LIN {X 0,Y 467.565,Z 337.401,A -85,B 0,C 180,E1 -7610.122,E2 -7610.122} C_VEL
LIN {X 0,Y 469.367,Z 346.484,A -85,B 0,C 180,E1 -7612.893,E2 -7612.893} C_VEL
LIN {X 0,Y 469.775,Z 350.018,A -85,B 0,C 180,E1 -7613.888,E2 -7613.888} C_VEL
LIN {X 0,Y 468.945,Z 363.418,A -85,B 0,C 180,E1 -7617.35,E2 -7617.35} C_VEL
LIN {X 0,Y 468.563,Z 374.519,A -85,B 0,C 180,E1 -7620.086,E2 -7620.086} C_VEL
LIN {X 0,Y 468.19,Z 387.799,A -85,B 0,C 180,E1 -7623.236,E2 -7623.236} C_VEL
LIN {X 0,Y 467.873,Z 401.533,A -85,B 0,C 180,E1 -7626.39,E2 -7626.39} C_VEL
LIN {X 0,Y 467.562,Z 416.649,A -85,B 0,C 180,E1 -7629.775,E2 -7629.775} C_VEL
LIN {X 0,Y 467.339,Z 431.071,A -85,B 0,C 180,E1 -7632.948,E2 -7632.948} C_VEL
LIN {X 0,Y 467.254,Z 438.483,A -85,B 0,C 180,E1 -7634.516,E2 -7634.516} C_VEL
LIN {X 0,Y 467.458,Z 441.247,A -85,B 0,C 180,E1 -7634.62,E2 -7634.62} C_VEL
LIN {X 0,Y 468.524,Z 455.112,A -85,B 0,C 180,E1 -7635.032,E2 -7635.032} C_VEL
LIN {X 0,Y 469.497,Z 465.721,A -85,B 0,C 180,E1 -7635.479,E2 -7635.479} C_VEL
LIN {X 0,Y 469.015,Z 478.326,A -85,B 0,C 180,E1 -7636.128,E2 -7636.128} C_VEL
LIN {X 0,Y 468.559,Z 489.635,A -85,B 0,C 180,E1 -7636.888,E2 -7636.888} C_VEL
LIN {X 0,Y 468.224,Z 499.908,A -85,B 0,C 180,E1 -7637.742,E2 -7637.742} C_VEL
LIN {X 0,Y 467.755,Z 509.75,A -85,B 0,C 180,E1 -7638.737,E2 -7638.737} C_VEL
LIN {X 0,Y 467.388,Z 518.626,A -85,B 0,C 180,E1 -7639.824,E2 -7639.824} C_VEL
LIN {X 0,Y 467.148,Z 527.303,A -85,B 0,C 180,E1 -7641.129,E2 -7641.129} C_VEL
LIN {X 0,Y 467.045,Z 534.318,A -85,B 0,C 180,E1 -7642.434,E2 -7642.434} C_VEL
LIN {X 0,Y 467.012,Z 540.786,A -85,B 0,C 180,E1 -7643.953,E2 -7643.953} C_VEL
LIN {X 0,Y 466.979,Z 544.992,A -85,B 0,C 180,E1 -7645.252,E2 -7645.252} C_VEL
LIN {X 0,Y 466.988,Z 548.116,A -85,B 0,C 180,E1 -7646.549,E2 -7646.549} C_VEL
LIN {X 0,Y 466.982,Z 549.617,A -85,B 0,C 180,E1 -7647.412,E2 -7647.412} C_VEL
LIN {X 0,Y 467.076,Z 551.385,A -85,B 0,C 180,E1 -7649.138,E2 -7649.138} C_VEL
LIN {X 0,Y 467.064,Z 551.647,A -85,B 0,C 180,E1 -7650,E2 -7650} C_VEL
LIN {X 0,Y 467.075,Z 551.459,A -85,B 0,C 180,E1 -7650.862,E2 -7650.862} C_VEL
LIN {X 0,Y 466.955,Z 549.855,A -85,B 0,C 180,E1 -7652.588,E2 -7652.588} C_VEL
LIN {X 0,Y 466.966,Z 548.427,A -85,B 0,C 180,E1 -7653.451,E2 -7653.451} C_VEL
LIN {X 0,Y 466.951,Z 545.43,A -85,B 0,C 180,E1 -7654.748,E2 -7654.748} C_VEL
LIN {X 0,Y 466.971,Z 540.24,A -85,B 0,C 180,E1 -7656.343,E2 -7656.343} C_VEL
LIN {X 0,Y 467.03,Z 534.045,A -85,B 0,C 180,E1 -7657.784,E2 -7657.784} C_VEL
LIN {X 0,Y 467.175,Z 526.937,A -85,B 0,C 180,E1 -7659.088,E2 -7659.088} C_VEL
LIN {X 0,Y 467.453,Z 518.079,A -85,B 0,C 180,E1 -7660.394,E2 -7660.394} C_VEL
LIN {X 0,Y 467.832,Z 509.046,A -85,B 0,C 180,E1 -7661.481,E2 -7661.481} C_VEL
LIN {X 0,Y 468.296,Z 499.714,A -85,B 0,C 180,E1 -7662.406,E2 -7662.406} C_VEL
LIN {X 0,Y 468.724,Z 488.228,A -85,B 0,C 180,E1 -7663.328,E2 -7663.328} C_VEL
LIN {X 0,Y 469.261,Z 476.177,A -85,B 0,C 180,E1 -7664.085,E2 -7664.085} C_VEL
LIN {X 0,Y 469.619,Z 464.972,A -85,B 0,C 180,E1 -7664.627,E2 -7664.627} C_VEL
LIN {X 0,Y 468.446,Z 452.922,A -85,B 0,C 180,E1 -7665.096,E2 -7665.096} C_VEL
LIN {X 0,Y 467.289,Z 441.274,A -85,B 0,C 180,E1 -7665.427,E2 -7665.427} C_VEL
LIN {X 0,Y 467.275,Z 440.651,A -85,B 0,C 180,E1 -7665.483,E2 -7665.483} C_VEL
LIN {X 0,Y 467.587,Z 425.096,A -85,B 0,C 180,E1 -7668.974,E2 -7668.974} C_VEL
LIN {X 0,Y 468,Z 409.645,A -85,B 0,C 180,E1 -7672.515,E2 -7672.515} C_VEL
LIN {X 0,Y 468.463,Z 395.511,A -85,B 0,C 180,E1 -7675.824,E2 -7675.824} C_VEL
LIN {X 0,Y 468.898,Z 382.637,A -85,B 0,C 180,E1 -7678.905,E2 -7678.905} C_VEL
LIN {X 0,Y 469.437,Z 370.623,A -85,B 0,C 180,E1 -7681.851,E2 -7681.851} C_VEL
LIN {X 0,Y 470.388,Z 355.622,A -85,B 0,C 180,E1 -7685.639,E2 -7685.639} C_VEL
LIN {X 0,Y 470.406,Z 351.582,A -85,B 0,C 180,E1 -7686.698,E2 -7686.698} C_VEL
LIN {X 0,Y 468.436,Z 341.626,A -85,B 0,C 180,E1 -7689.523,E2 -7689.523} C_VEL
LIN {X 0,Y 467.561,Z 337.324,A -85,B 0,C 180,E1 -7690.832,E2 -7690.832} C_VEL
LIN {X 0,Y 467.539,Z 337.249,A -85,B 0,C 180,E1 -7693.819,E2 -7693.819} C_VEL
LIN {X 0,Y 467.54,Z 337.245,A -85,B 0,C 180,E1 -7696.254,E2 -7696.254} C_VEL
LIN {X 0,Y 467.551,Z 337.244,A -85,B 0,C 180,E1 -7699.732,E2 -7699.732} C_VEL
LIN {X 0,Y 467.54,Z 337.244,A -85,B 0,C 180,E1 -7702.813,E2 -7702.813} C_VEL
LIN {X 0,Y 467.569,Z 337.24,A -85,B 0,C 180,E1 -7705.759,E2 -7705.759} C_VEL
LIN {X 0,Y 467.559,Z 337.243,A -85,B 0,C 180,E1 -7708.955,E2 -7708.955} C_VEL
LIN {X 0,Y 467.625,Z 337.232,A -85,B 0,C 180,E1 -7712.461,E2 -7712.461} C_VEL
LIN {X 0,Y 467.576,Z 337.245,A -85,B 0,C 180,E1 -7715.111,E2 -7715.111} C_VEL
LIN {X 0,Y 467.524,Z 337.244,A -85,B 0,C 180,E1 -7717.926,E2 -7717.926} C_VEL
LIN {X 0,Y 467.612,Z 337.236,A -85,B 0,C 180,E1 -7720.692,E2 -7720.692} C_VEL
LIN {X 0,Y 467.628,Z 337.231,A -85,B 0,C 180,E1 -7724.305,E2 -7724.305} C_VEL
LIN {X 0,Y 467.645,Z 337.228,A -85,B 0,C 180,E1 -7727.854,E2 -7727.854} C_VEL
LIN {X 0,Y 467.659,Z 337.229,A -85,B 0,C 180,E1 -7731.357,E2 -7731.357} C_VEL
LIN {X 0,Y 467.722,Z 337.219,A -85,B 0,C 180,E1 -7733.962,E2 -7733.962} C_VEL
LIN {X 0,Y 467.846,Z 337.205,A -85,B 0,C 180,E1 -7737.417,E2 -7737.417} C_VEL
LIN {X 0,Y 467.869,Z 337.201,A -85,B 0,C 180,E1 -7740,E2 -7740} C_VEL
LIN {X 0,Y 467.847,Z 337.209,A -85,B 0,C 180,E1 -7742.583,E2 -7742.583} C_VEL
LIN {X 0,Y 467.723,Z 337.22,A -85,B 0,C 180,E1 -7746.038,E2 -7746.038} C_VEL
LIN {X 0,Y 467.671,Z 337.233,A -85,B 0,C 180,E1 -7748.643,E2 -7748.643} C_VEL
LIN {X 0,Y 467.646,Z 337.231,A -85,B 0,C 180,E1 -7752.146,E2 -7752.146} C_VEL
LIN {X 0,Y 467.629,Z 337.23,A -85,B 0,C 180,E1 -7755.695,E2 -7755.695} C_VEL
LIN {X 0,Y 467.608,Z 337.238,A -85,B 0,C 180,E1 -7758.765,E2 -7758.765} C_VEL
LIN {X 0,Y 467.575,Z 337.238,A -85,B 0,C 180,E1 -7761.27,E2 -7761.27} C_VEL
LIN {X 0,Y 467.567,Z 337.24,A -85,B 0,C 180,E1 -7763.944,E2 -7763.944} C_VEL
LIN {X 0,Y 467.608,Z 337.236,A -85,B 0,C 180,E1 -7766.801,E2 -7766.801} C_VEL
LIN {X 0,Y 467.579,Z 337.238,A -85,B 0,C 180,E1 -7769.736,E2 -7769.736} C_VEL
LIN {X 0,Y 467.576,Z 337.24,A -85,B 0,C 180,E1 -7772.759,E2 -7772.759} C_VEL
LIN {X 0,Y 467.549,Z 337.243,A -85,B 0,C 180,E1 -7775.89,E2 -7775.89} C_VEL
LIN {X 0,Y 467.591,Z 337.235,A -85,B 0,C 180,E1 -7779.144,E2 -7779.144} C_VEL
LIN {X 0,Y 467.581,Z 337.24,A -85,B 0,C 180,E1 -7782.568,E2 -7782.568} C_VEL
LIN {X 0,Y 467.566,Z 337.238,A -85,B 0,C 180,E1 -7785.054,E2 -7785.054} C_VEL
LIN {X 0,Y 467.585,Z 337.237,A -85,B 0,C 180,E1 -7787.441,E2 -7787.441} C_VEL
LIN {X 0,Y 467.578,Z 337.237,A -85,B 0,C 180,E1 -7790.856,E2 -7790.856} C_VEL
LIN {X 0,Y 467.56,Z 337.244,A -85,B 0,C 180,E1 -7794.261,E2 -7794.261} C_VEL
LIN {X 0,Y 467.58,Z 337.237,A -85,B 0,C 180,E1 -7797.322,E2 -7797.322} C_VEL
LIN {X 0,Y 467.578,Z 337.237,A -85,B 0,C 180,E1 -7800.666,E2 -7800.666} C_VEL
LIN {X 0,Y 467.628,Z 337.231,A -85,B 0,C 180,E1 -7803.201,E2 -7803.201} C_VEL
LIN {X 0,Y 467.594,Z 337.236,A -85,B 0,C 180,E1 -7806.469,E2 -7806.469} C_VEL
LIN {X 0,Y 467.625,Z 337.239,A -85,B 0,C 180,E1 -7809.778,E2 -7809.778} C_VEL
LIN {X 0,Y 467.61,Z 337.233,A -85,B 0,C 180,E1 -7812.507,E2 -7812.507} C_VEL
LIN {X 0,Y 467.608,Z 337.235,A -85,B 0,C 180,E1 -7815.197,E2 -7815.197} C_VEL
LIN {X 0,Y 467.599,Z 337.235,A -85,B 0,C 180,E1 -7815.441,E2 -7815.441} C_VEL
LIN {X 0,Y 466.929,Z 337.321,A -85,B 0,C 180,E1 -7816.16,E2 -7816.16} C_VEL
LIN {X 0,Y 464.085,Z 337.675,A -85,B 0,C 180,E1 -7817.329,E2 -7817.329} C_VEL
LIN {X 0,Y 461.686,Z 337.972,A -85,B 0,C 180,E1 -7818.271,E2 -7818.271} C_VEL
LIN {X 0,Y 460.661,Z 338.099,A -85,B 0,C 180,E1 -7818.998,E2 -7818.998} C_VEL
LIN {X 0,Y 460.58,Z 338.111,A -85,B 0,C 180,E1 -7819.245,E2 -7819.245} C_VEL
LIN {X 0,Y 460.723,Z 338.091,A -85,B 0,C 180,E1 -7822.538,E2 -7822.538} C_VEL
LIN {X 0,Y 460.702,Z 338.093,A -85,B 0,C 180,E1 -7824.749,E2 -7824.749} C_VEL
LIN {X 0,Y 460.828,Z 338.083,A -85,B 0,C 180,E1 -7827.378,E2 -7827.378} C_VEL
LIN {X 0,Y 460.857,Z 338.077,A -85,B 0,C 180,E1 -7830,E2 -7830} C_VEL
LIN {X 0,Y 460.828,Z 338.078,A -85,B 0,C 180,E1 -7832.622,E2 -7832.622} C_VEL
LIN {X 0,Y 460.704,Z 338.094,A -85,B 0,C 180,E1 -7836.13,E2 -7836.13} C_VEL
LIN {X 0,Y 460.631,Z 338.103,A -85,B 0,C 180,E1 -7838.776,E2 -7838.776} C_VEL
LIN {X 0,Y 460.615,Z 338.104,A -85,B 0,C 180,E1 -7842.445,E2 -7842.445} C_VEL
LIN {X 0,Y 460.602,Z 338.107,A -85,B 0,C 180,E1 -7845.997,E2 -7845.997} C_VEL
LIN {X 0,Y 460.573,Z 338.113,A -85,B 0,C 180,E1 -7848.902,E2 -7848.902} C_VEL
LIN {X 0,Y 460.517,Z 338.121,A -85,B 0,C 180,E1 -7851.485,E2 -7851.485} C_VEL
LIN {X 0,Y 460.543,Z 338.113,A -85,B 0,C 180,E1 -7854.332,E2 -7854.332} C_VEL
LIN {X 0,Y 460.584,Z 338.115,A -85,B 0,C 180,E1 -7857.242,E2 -7857.242} C_VEL
LIN {X 0,Y 460.51,Z 338.117,A -85,B 0,C 180,E1 -7860.239,E2 -7860.239} C_VEL
LIN {X 0,Y 460.528,Z 338.12,A -85,B 0,C 180,E1 -7863.324,E2 -7863.324} C_VEL
LIN {X 0,Y 460.479,Z 338.123,A -85,B 0,C 180,E1 -7866.528,E2 -7866.528} C_VEL
LIN {X 0,Y 460.576,Z 338.111,A -85,B 0,C 180,E1 -7869.857,E2 -7869.857} C_VEL
LIN {X 0,Y 460.539,Z 338.121,A -85,B 0,C 180,E1 -7872.904,E2 -7872.904} C_VEL
LIN {X 0,Y 460.519,Z 338.121,A -85,B 0,C 180,E1 -7875.828,E2 -7875.828} C_VEL
LIN {X 0,Y 460.635,Z 338.281,A -85,B 0,C 180,E1 -7877.236,E2 -7877.236} C_VEL
LIN {X 0,Y 460.785,Z 339.139,A -85,B 0,C 180,E1 -7877.371,E2 -7877.371} C_VEL
LIN {X 0,Y 463.382,Z 348.732,A -85,B 0,C 180,E1 -7878.001,E2 -7878.001} C_VEL
LIN {X 0,Y 462.957,Z 360.559,A -85,B 0,C 180,E1 -7878.817,E2 -7878.817} C_VEL
LIN {X 0,Y 462.47,Z 371.478,A -85,B 0,C 180,E1 -7879.77,E2 -7879.77} C_VEL
LIN {X 0,Y 462.064,Z 381.585,A -85,B 0,C 180,E1 -7880.868,E2 -7880.868} C_VEL
LIN {X 0,Y 461.625,Z 389.546,A -85,B 0,C 180,E1 -7881.923,E2 -7881.923} C_VEL
LIN {X 0,Y 461.224,Z 397.793,A -85,B 0,C 180,E1 -7883.267,E2 -7883.267} C_VEL
LIN {X 0,Y 460.926,Z 404.327,A -85,B 0,C 180,E1 -7884.591,E2 -7884.591} C_VEL
LIN {X 0,Y 460.623,Z 410.341,A -85,B 0,C 180,E1 -7886.158,E2 -7886.158} C_VEL
LIN {X 0,Y 460.442,Z 414.737,A -85,B 0,C 180,E1 -7887.709,E2 -7887.709} C_VEL
LIN {X 0,Y 460.369,Z 416.902,A -85,B 0,C 180,E1 -7888.746,E2 -7888.746} C_VEL
LIN {X 0,Y 460.222,Z 419.248,A -85,B 0,C 180,E1 -7890.507,E2 -7890.507} C_VEL
LIN {X 0,Y 460.209,Z 419.967,A -85,B 0,C 180,E1 -7892.34,E2 -7892.34} C_VEL
LIN {X 0,Y 460.319,Z 418.895,A -85,B 0,C 180,E1 -7894.26,E2 -7894.26} C_VEL
LIN {X 0,Y 460.457,Z 416.885,A -85,B 0,C 180,E1 -7895.663,E2 -7895.663} C_VEL
LIN {X 0,Y 460.657,Z 413.689,A -85,B 0,C 180,E1 -7897.105,E2 -7897.105} C_VEL
LIN {X 0,Y 460.883,Z 409.313,A -85,B 0,C 180,E1 -7898.532,E2 -7898.532} C_VEL
LIN {X 0,Y 461.218,Z 403.626,A -85,B 0,C 180,E1 -7899.949,E2 -7899.949} C_VEL
LIN {X 0,Y 461.631,Z 396.366,A -85,B 0,C 180,E1 -7901.355,E2 -7901.355} C_VEL
LIN {X 0,Y 462.119,Z 387.293,A -85,B 0,C 180,E1 -7902.749,E2 -7902.749} C_VEL
LIN {X 0,Y 462.661,Z 377.58,A -85,B 0,C 180,E1 -7903.926,E2 -7903.926} C_VEL
LIN {X 0,Y 463.097,Z 367.275,A -85,B 0,C 180,E1 -7904.936,E2 -7904.936} C_VEL
LIN {X 0,Y 463.511,Z 356.547,A -85,B 0,C 180,E1 -7905.779,E2 -7905.779} C_VEL
LIN {X 0,Y 463.584,Z 348.504,A -85,B 0,C 180,E1 -7906.298,E2 -7906.298} C_VEL
LIN {X 0,Y 460.717,Z 338.858,A -85,B 0,C 180,E1 -7906.958,E2 -7906.958} C_VEL
LIN {X 0,Y 460.583,Z 338.152,A -85,B 0,C 180,E1 -7907.139,E2 -7907.139} C_VEL
LIN {X 0,Y 460.577,Z 338.116,A -85,B 0,C 180,E1 -7909.449,E2 -7909.449} C_VEL
LIN {X 0,Y 460.704,Z 338.097,A -85,B 0,C 180,E1 -7912.543,E2 -7912.543} C_VEL
LIN {X 0,Y 460.682,Z 338.101,A -85,B 0,C 180,E1 -7914.748,E2 -7914.748} C_VEL
LIN {X 0,Y 460.788,Z 338.089,A -85,B 0,C 180,E1 -7917.377,E2 -7917.377} C_VEL
LIN {X 0,Y 460.84,Z 338.079,A -85,B 0,C 180,E1 -7920,E2 -7920} C_VEL
LIN {X 0,Y 460.788,Z 338.086,A -85,B 0,C 180,E1 -7922.623,E2 -7922.623} C_VEL
LIN {X 0,Y 460.687,Z 338.097,A -85,B 0,C 180,E1 -7926.13,E2 -7926.13} C_VEL
LIN {X 0,Y 460.609,Z 338.109,A -85,B 0,C 180,E1 -7928.777,E2 -7928.777} C_VEL
LIN {X 0,Y 460.598,Z 338.107,A -85,B 0,C 180,E1 -7932.335,E2 -7932.335} C_VEL
LIN {X 0,Y 460.591,Z 338.109,A -85,B 0,C 180,E1 -7935.998,E2 -7935.998} C_VEL
LIN {X 0,Y 460.558,Z 338.113,A -85,B 0,C 180,E1 -7939.616,E2 -7939.616} C_VEL
LIN {X 0,Y 460.501,Z 338.122,A -85,B 0,C 180,E1 -7942.429,E2 -7942.429} C_VEL
LIN {X 0,Y 460.545,Z 338.113,A -85,B 0,C 180,E1 -7945.799,E2 -7945.799} C_VEL
LIN {X 0,Y 460.543,Z 338.116,A -85,B 0,C 180,E1 -7948.234,E2 -7948.234} C_VEL
LIN {X 0,Y 460.512,Z 338.122,A -85,B 0,C 180,E1 -7951.283,E2 -7951.283} C_VEL
LIN {X 0,Y 460.515,Z 338.122,A -85,B 0,C 180,E1 -7954.504,E2 -7954.504} C_VEL
LIN {X 0,Y 460.493,Z 338.123,A -85,B 0,C 180,E1 -7957.624,E2 -7957.624} C_VEL
LIN {X 0,Y 460.509,Z 338.124,A -85,B 0,C 180,E1 -7961.014,E2 -7961.014} C_VEL
LIN {X 0,Y 460.506,Z 338.121,A -85,B 0,C 180,E1 -7964.59,E2 -7964.59} C_VEL
LIN {X 0,Y 460.486,Z 338.124,A -85,B 0,C 180,E1 -7967.816,E2 -7967.816} C_VEL
LIN {X 0,Y 460.534,Z 338.278,A -85,B 0,C 180,E1 -7969.808,E2 -7969.808} C_VEL
LIN {X 0,Y 462.265,Z 347.022,A -85,B 0,C 180,E1 -7972.546,E2 -7972.546} C_VEL
LIN {X 0,Y 462.809,Z 350.922,A -85,B 0,C 180,E1 -7973.685,E2 -7973.685} C_VEL
LIN {X 0,Y 462.069,Z 362.679,A -85,B 0,C 180,E1 -7976.802,E2 -7976.802} C_VEL
LIN {X 0,Y 461.581,Z 374.697,A -85,B 0,C 180,E1 -7979.838,E2 -7979.838} C_VEL
LIN {X 0,Y 461.162,Z 387.905,A -85,B 0,C 180,E1 -7983.04,E2 -7983.04} C_VEL
LIN {X 0,Y 460.8,Z 401.493,A -85,B 0,C 180,E1 -7986.221,E2 -7986.221} C_VEL
LIN {X 0,Y 460.528,Z 415.613,A -85,B 0,C 180,E1 -7989.452,E2 -7989.452} C_VEL
LIN {X 0,Y 460.278,Z 429.983,A -85,B 0,C 180,E1 -7992.678,E2 -7992.678} C_VEL
LIN {X 0,Y 460.201,Z 437.169,A -85,B 0,C 180,E1 -7994.239,E2 -7994.239} C_VEL
LIN {X 0,Y 460.353,Z 439.549,A -85,B 0,C 180,E1 -7994.356,E2 -7994.356} C_VEL
LIN {X 0,Y 461.551,Z 454.098,A -85,B 0,C 180,E1 -7994.798,E2 -7994.798} C_VEL
LIN {X 0,Y 462.484,Z 467.088,A -85,B 0,C 180,E1 -7995.367,E2 -7995.367} C_VEL
LIN {X 0,Y 461.995,Z 478.993,A -85,B 0,C 180,E1 -7996.026,E2 -7996.026} C_VEL
LIN {X 0,Y 461.521,Z 489.961,A -85,B 0,C 180,E1 -7996.796,E2 -7996.796} C_VEL
LIN {X 0,Y 461.166,Z 500.175,A -85,B 0,C 180,E1 -7997.681,E2 -7997.681} C_VEL
LIN {X 0,Y 460.677,Z 508.638,A -85,B 0,C 180,E1 -7998.561,E2 -7998.561} C_VEL
LIN {X 0,Y 460.329,Z 517.532,A -85,B 0,C 180,E1 -7999.666,E2 -7999.666} C_VEL
LIN {X 0,Y 460.093,Z 526.222,A -85,B 0,C 180,E1 -8000.992,E2 -8000.992} C_VEL
LIN {X 0,Y 459.988,Z 533.25,A -85,B 0,C 180,E1 -8002.317,E2 -8002.317} C_VEL
LIN {X 0,Y 459.957,Z 539.734,A -85,B 0,C 180,E1 -8003.86,E2 -8003.86} C_VEL
LIN {X 0,Y 459.935,Z 543.956,A -85,B 0,C 180,E1 -8005.179,E2 -8005.179} C_VEL
LIN {X 0,Y 459.943,Z 547.093,A -85,B 0,C 180,E1 -8006.496,E2 -8006.496} C_VEL
LIN {X 0,Y 459.941,Z 548.602,A -85,B 0,C 180,E1 -8007.373,E2 -8007.373} C_VEL
LIN {X 0,Y 460.058,Z 550.388,A -85,B 0,C 180,E1 -8009.125,E2 -8009.125} C_VEL
LIN {X 0,Y 460.047,Z 550.654,A -85,B 0,C 180,E1 -8010,E2 -8010} C_VEL
LIN {X 0,Y 460.055,Z 550.469,A -85,B 0,C 180,E1 -8010.875,E2 -8010.875} C_VEL
LIN {X 0,Y 459.911,Z 548.868,A -85,B 0,C 180,E1 -8012.628,E2 -8012.628} C_VEL
LIN {X 0,Y 459.922,Z 547.439,A -85,B 0,C 180,E1 -8013.504,E2 -8013.504} C_VEL
LIN {X 0,Y 459.901,Z 544.441,A -85,B 0,C 180,E1 -8014.821,E2 -8014.821} C_VEL
LIN {X 0,Y 459.916,Z 540.361,A -85,B 0,C 180,E1 -8016.14,E2 -8016.14} C_VEL
LIN {X 0,Y 459.944,Z 534.065,A -85,B 0,C 180,E1 -8017.683,E2 -8017.683} C_VEL
LIN {X 0,Y 460.062,Z 527.212,A -85,B 0,C 180,E1 -8019.008,E2 -8019.008} C_VEL
LIN {X 0,Y 460.33,Z 518.695,A -85,B 0,C 180,E1 -8020.334,E2 -8020.334} C_VEL
LIN {X 0,Y 460.702,Z 509.962,A -85,B 0,C 180,E1 -8021.438,E2 -8021.438} C_VEL
LIN {X 0,Y 461.229,Z 499.913,A -85,B 0,C 180,E1 -8022.48,E2 -8022.48} C_VEL
LIN {X 0,Y 461.684,Z 488.694,A -85,B 0,C 180,E1 -8023.423,E2 -8023.423} C_VEL
LIN {X 0,Y 462.225,Z 476.992,A -85,B 0,C 180,E1 -8024.192,E2 -8024.192} C_VEL
LIN {X 0,Y 462.592,Z 465.049,A -85,B 0,C 180,E1 -8024.798,E2 -8024.798} C_VEL
LIN {X 0,Y 461.533,Z 453.855,A -85,B 0,C 180,E1 -8025.256,E2 -8025.256} C_VEL
LIN {X 0,Y 460.207,Z 440.092,A -85,B 0,C 180,E1 -8025.681,E2 -8025.681} C_VEL
LIN {X 0,Y 460.253,Z 434.646,A -85,B 0,C 180,E1 -8026.865,E2 -8026.865} C_VEL
LIN {X 0,Y 460.563,Z 422.734,A -85,B 0,C 180,E1 -8029.615,E2 -8029.615} C_VEL
LIN {X 0,Y 460.978,Z 408.837,A -85,B 0,C 180,E1 -8032.877,E2 -8032.877} C_VEL
LIN {X 0,Y 461.47,Z 394.863,A -85,B 0,C 180,E1 -8036.209,E2 -8036.209} C_VEL
LIN {X 0,Y 462.009,Z 381.331,A -85,B 0,C 180,E1 -8039.517,E2 -8039.517} C_VEL
LIN {X 0,Y 462.607,Z 368.871,A -85,B 0,C 180,E1 -8042.637,E2 -8042.637} C_VEL
LIN {X 0,Y 463.442,Z 356.88,A -85,B 0,C 180,E1 -8045.72,E2 -8045.72} C_VEL
LIN {X 0,Y 463.401,Z 352.544,A -85,B 0,C 180,E1 -8046.888,E2 -8046.888} C_VEL
LIN {X 0,Y 461.393,Z 342.566,A -85,B 0,C 180,E1 -8049.772,E2 -8049.772} C_VEL
LIN {X 0,Y 460.538,Z 338.198,A -85,B 0,C 180,E1 -8051.129,E2 -8051.129} C_VEL
LIN {X 0,Y 460.506,Z 338.122,A -85,B 0,C 180,E1 -8054.588,E2 -8054.588} C_VEL
LIN {X 0,Y 460.484,Z 338.124,A -85,B 0,C 180,E1 -8057.814,E2 -8057.814} C_VEL
LIN {X 0,Y 460.506,Z 338.118,A -85,B 0,C 180,E1 -8060.135,E2 -8060.135} C_VEL
LIN {X 0,Y 460.468,Z 338.128,A -85,B 0,C 180,E1 -8063.47,E2 -8063.47} C_VEL
LIN {X 0,Y 460.512,Z 338.118,A -85,B 0,C 180,E1 -8066.674,E2 -8066.674} C_VEL
LIN {X 0,Y 460.501,Z 338.12,A -85,B 0,C 180,E1 -8069.759,E2 -8069.759} C_VEL
LIN {X 0,Y 460.563,Z 338.113,A -85,B 0,C 180,E1 -8072.755,E2 -8072.755} C_VEL
LIN {X 0,Y 460.52,Z 338.118,A -85,B 0,C 180,E1 -8075.666,E2 -8075.666} C_VEL
LIN {X 0,Y 460.512,Z 338.119,A -85,B 0,C 180,E1 -8078.578,E2 -8078.578} C_VEL
LIN {X 0,Y 460.576,Z 338.114,A -85,B 0,C 180,E1 -8081.31,E2 -8081.31} C_VEL
LIN {X 0,Y 460.594,Z 338.107,A -85,B 0,C 180,E1 -8084.059,E2 -8084.059} C_VEL
LIN {X 0,Y 460.598,Z 338.107,A -85,B 0,C 180,E1 -8087.665,E2 -8087.665} C_VEL
LIN {X 0,Y 460.609,Z 338.109,A -85,B 0,C 180,E1 -8091.223,E2 -8091.223} C_VEL
LIN {X 0,Y 460.687,Z 338.095,A -85,B 0,C 180,E1 -8093.87,E2 -8093.87} C_VEL
LIN {X 0,Y 460.788,Z 338.084,A -85,B 0,C 180,E1 -8097.377,E2 -8097.377} C_VEL
LIN {X 0,Y 460.84,Z 338.076,A -85,B 0,C 180,E1 -8100,E2 -8100} C_VEL
LIN {X 0,Y 460.788,Z 338.089,A -85,B 0,C 180,E1 -8102.623,E2 -8102.623} C_VEL
LIN {X 0,Y 460.69,Z 338.096,A -85,B 0,C 180,E1 -8106.13,E2 -8106.13} C_VEL
LIN {X 0,Y 460.618,Z 338.111,A -85,B 0,C 180,E1 -8108.776,E2 -8108.776} C_VEL
LIN {X 0,Y 460.603,Z 338.111,A -85,B 0,C 180,E1 -8112.445,E2 -8112.445} C_VEL
LIN {X 0,Y 460.59,Z 338.109,A -85,B 0,C 180,E1 -8115.998,E2 -8115.998} C_VEL
LIN {X 0,Y 460.562,Z 338.114,A -85,B 0,C 180,E1 -8118.902,E2 -8118.902} C_VEL
LIN {X 0,Y 460.51,Z 338.117,A -85,B 0,C 180,E1 -8121.486,E2 -8121.486} C_VEL
LIN {X 0,Y 460.535,Z 338.12,A -85,B 0,C 180,E1 -8124.333,E2 -8124.333} C_VEL
LIN {X 0,Y 460.565,Z 338.111,A -85,B 0,C 180,E1 -8127.244,E2 -8127.244} C_VEL
LIN {X 0,Y 460.519,Z 338.122,A -85,B 0,C 180,E1 -8130.239,E2 -8130.239} C_VEL
LIN {X 0,Y 460.522,Z 338.116,A -85,B 0,C 180,E1 -8133.326,E2 -8133.326} C_VEL
LIN {X 0,Y 460.471,Z 338.127,A -85,B 0,C 180,E1 -8136.53,E2 -8136.53} C_VEL
LIN {X 0,Y 460.567,Z 338.113,A -85,B 0,C 180,E1 -8139.859,E2 -8139.859} C_VEL
LIN {X 0,Y 460.508,Z 338.118,A -85,B 0,C 180,E1 -8142.901,E2 -8142.901} C_VEL
LIN {X 0,Y 460.515,Z 338.12,A -85,B 0,C 180,E1 -8145.83,E2 -8145.83} C_VEL
LIN {X 0,Y 460.53,Z 338.115,A -85,B 0,C 180,E1 -8148.99,E2 -8148.99} C_VEL
LIN {X 0,Y 460.523,Z 338.116,A -85,B 0,C 180,E1 -8151.268,E2 -8151.268} C_VEL
LIN {X 0,Y 460.511,Z 338.119,A -85,B 0,C 180,E1 -8154.555,E2 -8154.555} C_VEL
LIN {X 0,Y 460.53,Z 338.119,A -85,B 0,C 180,E1 -8157.716,E2 -8157.716} C_VEL
LIN {X 0,Y 460.547,Z 338.113,A -85,B 0,C 180,E1 -8160.77,E2 -8160.77} C_VEL
LIN {X 0,Y 460.568,Z 338.116,A -85,B 0,C 180,E1 -8163.736,E2 -8163.736} C_VEL
LIN {X 0,Y 460.547,Z 338.113,A -85,B 0,C 180,E1 -8166.625,E2 -8166.625} C_VEL
LIN {X 0,Y 460.553,Z 338.115,A -85,B 0,C 180,E1 -8169.453,E2 -8169.453} C_VEL
LIN {X 0,Y 460.561,Z 338.114,A -85,B 0,C 180,E1 -8172.231,E2 -8172.231} C_VEL
LIN {X 0,Y 460.571,Z 338.11,A -85,B 0,C 180,E1 -8174.965,E2 -8174.965} C_VEL
LIN {X 0,Y 460.614,Z 338.104,A -85,B 0,C 180,E1 -8178.56,E2 -8178.56} C_VEL
LIN {X 0,Y 460.58,Z 338.111,A -85,B 0,C 180,E1 -8179.245,E2 -8179.245} C_VEL
LIN {X 0,Y 459.926,Z 338.198,A -85,B 0,C 180,E1 -8179.975,E2 -8179.975} C_VEL
LIN {X 0,Y 457.108,Z 338.547,A -85,B 0,C 180,E1 -8181.162,E2 -8181.162} C_VEL
LIN {X 0,Y 454.729,Z 338.84,A -85,B 0,C 180,E1 -8182.119,E2 -8182.119} C_VEL
LIN {X 0,Y 453.718,Z 338.964,A -85,B 0,C 180,E1 -8182.858,E2 -8182.858} C_VEL
LIN {X 0,Y 453.641,Z 338.974,A -85,B 0,C 180,E1 -8183.108,E2 -8183.108} C_VEL
LIN {X 0,Y 453.676,Z 338.969,A -85,B 0,C 180,E1 -8184.667,E2 -8184.667} C_VEL
LIN {X 0,Y 453.768,Z 338.962,A -85,B 0,C 180,E1 -8187.337,E2 -8187.337} C_VEL
LIN {X 0,Y 453.827,Z 338.952,A -85,B 0,C 180,E1 -8190,E2 -8190} C_VEL
LIN {X 0,Y 453.769,Z 338.957,A -85,B 0,C 180,E1 -8192.663,E2 -8192.663} C_VEL
LIN {X 0,Y 453.672,Z 338.969,A -85,B 0,C 180,E1 -8196.225,E2 -8196.225} C_VEL
LIN {X 0,Y 453.595,Z 338.981,A -85,B 0,C 180,E1 -8198.913,E2 -8198.913} C_VEL
LIN {X 0,Y 453.565,Z 338.983,A -85,B 0,C 180,E1 -8202.528,E2 -8202.528} C_VEL
LIN {X 0,Y 453.546,Z 338.985,A -85,B 0,C 180,E1 -8206.195,E2 -8206.195} C_VEL
LIN {X 0,Y 453.522,Z 338.993,A -85,B 0,C 180,E1 -8209.041,E2 -8209.041} C_VEL
LIN {X 0,Y 453.478,Z 338.995,A -85,B 0,C 180,E1 -8211.835,E2 -8211.835} C_VEL
LIN {X 0,Y 453.515,Z 338.991,A -85,B 0,C 180,E1 -8214.734,E2 -8214.734} C_VEL
LIN {X 0,Y 453.537,Z 338.986,A -85,B 0,C 180,E1 -8217.96,E2 -8217.96} C_VEL
LIN {X 0,Y 453.465,Z 338.998,A -85,B 0,C 180,E1 -8221.525,E2 -8221.525} C_VEL
LIN {X 0,Y 453.487,Z 338.996,A -85,B 0,C 180,E1 -8224.777,E2 -8224.777} C_VEL
LIN {X 0,Y 453.483,Z 338.993,A -85,B 0,C 180,E1 -8228.309,E2 -8228.309} C_VEL
LIN {X 0,Y 453.513,Z 338.995,A -85,B 0,C 180,E1 -8230.606,E2 -8230.606} C_VEL
LIN {X 0,Y 453.478,Z 338.999,A -85,B 0,C 180,E1 -8233.247,E2 -8233.247} C_VEL
LIN {X 0,Y 453.554,Z 339.027,A -85,B 0,C 180,E1 -8236.941,E2 -8236.941} C_VEL
LIN {X 0,Y 453.744,Z 339.888,A -85,B 0,C 180,E1 -8237.142,E2 -8237.142} C_VEL
LIN {X 0,Y 456.329,Z 349.194,A -85,B 0,C 180,E1 -8237.77,E2 -8237.77} C_VEL
LIN {X 0,Y 456.168,Z 359.923,A -85,B 0,C 180,E1 -8238.51,E2 -8238.51} C_VEL
LIN {X 0,Y 455.615,Z 371.496,A -85,B 0,C 180,E1 -8239.512,E2 -8239.512} C_VEL
LIN {X 0,Y 455.212,Z 380.943,A -85,B 0,C 180,E1 -8240.527,E2 -8240.527} C_VEL
LIN {X 0,Y 454.768,Z 388.743,A -85,B 0,C 180,E1 -8241.536,E2 -8241.536} C_VEL
LIN {X 0,Y 454.353,Z 397.354,A -85,B 0,C 180,E1 -8242.896,E2 -8242.896} C_VEL
LIN {X 0,Y 453.997,Z 404.151,A -85,B 0,C 180,E1 -8244.241,E2 -8244.241} C_VEL
LIN {X 0,Y 453.671,Z 409.754,A -85,B 0,C 180,E1 -8245.627,E2 -8245.627} C_VEL
LIN {X 0,Y 453.459,Z 414.481,A -85,B 0,C 180,E1 -8247.149,E2 -8247.149} C_VEL
LIN {X 0,Y 453.378,Z 417.5,A -85,B 0,C 180,E1 -8248.491,E2 -8248.491} C_VEL
LIN {X 0,Y 453.295,Z 418.758,A -85,B 0,C 180,E1 -8249.227,E2 -8249.227} C_VEL
LIN {X 0,Y 453.231,Z 420.019,A -85,B 0,C 180,E1 -8250.266,E2 -8250.266} C_VEL
LIN {X 0,Y 453.196,Z 420.772,A -85,B 0,C 180,E1 -8251.266,E2 -8251.266} C_VEL
LIN {X 0,Y 453.197,Z 420.984,A -85,B 0,C 180,E1 -8252.275,E2 -8252.275} C_VEL
LIN {X 0,Y 453.28,Z 420.165,A -85,B 0,C 180,E1 -8254.06,E2 -8254.06} C_VEL
LIN {X 0,Y 453.376,Z 418.692,A -85,B 0,C 180,E1 -8255.257,E2 -8255.257} C_VEL
LIN {X 0,Y 453.594,Z 415.875,A -85,B 0,C 180,E1 -8256.728,E2 -8256.728} C_VEL
LIN {X 0,Y 453.857,Z 411.55,A -85,B 0,C 180,E1 -8258.292,E2 -8258.292} C_VEL
LIN {X 0,Y 454.242,Z 405.592,A -85,B 0,C 180,E1 -8259.864,E2 -8259.864} C_VEL
LIN {X 0,Y 454.682,Z 398.628,A -85,B 0,C 180,E1 -8261.293,E2 -8261.293} C_VEL
LIN {X 0,Y 455.086,Z 391.457,A -85,B 0,C 180,E1 -8262.474,E2 -8262.474} C_VEL
LIN {X 0,Y 455.619,Z 382.266,A -85,B 0,C 180,E1 -8263.701,E2 -8263.701} C_VEL
LIN {X 0,Y 456.148,Z 371.935,A -85,B 0,C 180,E1 -8264.816,E2 -8264.816} C_VEL
LIN {X 0,Y 456.593,Z 361.11,A -85,B 0,C 180,E1 -8265.743,E2 -8265.743} C_VEL
LIN {X 0,Y 456.968,Z 351.18,A -85,B 0,C 180,E1 -8266.424,E2 -8266.424} C_VEL
LIN {X 0,Y 454.239,Z 341.525,A -85,B 0,C 180,E1 -8267.087,E2 -8267.087} C_VEL
LIN {X 0,Y 453.662,Z 339.698,A -85,B 0,C 180,E1 -8267.227,E2 -8267.227} C_VEL
LIN {X 0,Y 453.592,Z 339.006,A -85,B 0,C 180,E1 -8267.449,E2 -8267.449} C_VEL
LIN {X 0,Y 453.582,Z 338.986,A -85,B 0,C 180,E1 -8271.086,E2 -8271.086} C_VEL
LIN {X 0,Y 453.658,Z 338.977,A -85,B 0,C 180,E1 -8273.774,E2 -8273.774} C_VEL
LIN {X 0,Y 453.732,Z 338.967,A -85,B 0,C 180,E1 -8277.337,E2 -8277.337} C_VEL
LIN {X 0,Y 453.811,Z 338.955,A -85,B 0,C 180,E1 -8280,E2 -8280} C_VEL
LIN {X 0,Y 453.732,Z 338.965,A -85,B 0,C 180,E1 -8282.663,E2 -8282.663} C_VEL
LIN {X 0,Y 453.654,Z 338.973,A -85,B 0,C 180,E1 -8286.226,E2 -8286.226} C_VEL
LIN {X 0,Y 453.575,Z 338.986,A -85,B 0,C 180,E1 -8288.914,E2 -8288.914} C_VEL
LIN {X 0,Y 453.554,Z 338.986,A -85,B 0,C 180,E1 -8292.529,E2 -8292.529} C_VEL
LIN {X 0,Y 453.535,Z 338.988,A -85,B 0,C 180,E1 -8296.196,E2 -8296.196} C_VEL
LIN {X 0,Y 453.507,Z 338.997,A -85,B 0,C 180,E1 -8299.04,E2 -8299.04} C_VEL
LIN {X 0,Y 453.467,Z 338.997,A -85,B 0,C 180,E1 -8301.837,E2 -8301.837} C_VEL
LIN {X 0,Y 453.495,Z 338.996,A -85,B 0,C 180,E1 -8304.736,E2 -8304.736} C_VEL
LIN {X 0,Y 453.523,Z 338.99,A -85,B 0,C 180,E1 -8307.96,E2 -8307.96} C_VEL
LIN {X 0,Y 453.457,Z 338.999,A -85,B 0,C 180,E1 -8311.525,E2 -8311.525} C_VEL
LIN {X 0,Y 453.475,Z 339.001,A -85,B 0,C 180,E1 -8314.777,E2 -8314.777} C_VEL
LIN {X 0,Y 453.451,Z 339.002,A -85,B 0,C 180,E1 -8318.313,E2 -8318.313} C_VEL
LIN {X 0,Y 453.464,Z 339.002,A -85,B 0,C 180,E1 -8320.612,E2 -8320.612} C_VEL
LIN {X 0,Y 453.453,Z 339,A -85,B 0,C 180,E1 -8324.223,E2 -8324.223} C_VEL
LIN {X 0,Y 453.432,Z 339.006,A -85,B 0,C 180,E1 -8327.003,E2 -8327.003} C_VEL
LIN {X 0,Y 453.515,Z 339.171,A -85,B 0,C 180,E1 -8329.487,E2 -8329.487} C_VEL
LIN {X 0,Y 455.362,Z 348.56,A -85,B 0,C 180,E1 -8332.501,E2 -8332.501} C_VEL
LIN {X 0,Y 455.878,Z 352.713,A -85,B 0,C 180,E1 -8333.729,E2 -8333.729} C_VEL
LIN {X 0,Y 454.985,Z 365.899,A -85,B 0,C 180,E1 -8337.274,E2 -8337.274} C_VEL
LIN {X 0,Y 454.465,Z 377.897,A -85,B 0,C 180,E1 -8340.34,E2 -8340.34} C_VEL
LIN {X 0,Y 454.107,Z 389.038,A -85,B 0,C 180,E1 -8343.084,E2 -8343.084} C_VEL
LIN {X 0,Y 453.719,Z 402.296,A -85,B 0,C 180,E1 -8346.251,E2 -8346.251} C_VEL
LIN {X 0,Y 453.416,Z 416.626,A -85,B 0,C 180,E1 -8349.59,E2 -8349.59} C_VEL
LIN {X 0,Y 453.153,Z 430.944,A -85,B 0,C 180,E1 -8352.863,E2 -8352.863} C_VEL
LIN {X 0,Y 453.104,Z 436.031,A -85,B 0,C 180,E1 -8353.974,E2 -8353.974} C_VEL
LIN {X 0,Y 453.28,Z 438.162,A -85,B 0,C 180,E1 -8354.08,E2 -8354.08} C_VEL
LIN {X 0,Y 454.553,Z 453.149,A -85,B 0,C 180,E1 -8354.554,E2 -8354.554} C_VEL
LIN {X 0,Y 455.399,Z 464.958,A -85,B 0,C 180,E1 -8355.077,E2 -8355.077} C_VEL
LIN {X 0,Y 455.257,Z 474.348,A -85,B 0,C 180,E1 -8355.586,E2 -8355.586} C_VEL
LIN {X 0,Y 454.654,Z 486.04,A -85,B 0,C 180,E1 -8356.366,E2 -8356.366} C_VEL
LIN {X 0,Y 454.124,Z 497.219,A -85,B 0,C 180,E1 -8357.308,E2 -8357.308} C_VEL
LIN {X 0,Y 453.761,Z 505.579,A -85,B 0,C 180,E1 -8358.158,E2 -8358.158} C_VEL
LIN {X 0,Y 453.411,Z 514.793,A -85,B 0,C 180,E1 -8359.281,E2 -8359.281} C_VEL
LIN {X 0,Y 453.099,Z 523.853,A -85,B 0,C 180,E1 -8360.627,E2 -8360.627} C_VEL
LIN {X 0,Y 452.939,Z 531.134,A -85,B 0,C 180,E1 -8361.973,E2 -8361.973} C_VEL
LIN {X 0,Y 452.865,Z 537.018,A -85,B 0,C 180,E1 -8363.324,E2 -8363.324} C_VEL
LIN {X 0,Y 452.861,Z 541.611,A -85,B 0,C 180,E1 -8364.657,E2 -8364.657} C_VEL
LIN {X 0,Y 452.894,Z 545.118,A -85,B 0,C 180,E1 -8365.996,E2 -8365.996} C_VEL
LIN {X 0,Y 452.898,Z 547.59,A -85,B 0,C 180,E1 -8367.332,E2 -8367.332} C_VEL
LIN {X 0,Y 453.037,Z 549.39,A -85,B 0,C 180,E1 -8369.111,E2 -8369.111} C_VEL
LIN {X 0,Y 453.028,Z 549.659,A -85,B 0,C 180,E1 -8370,E2 -8370} C_VEL
LIN {X 0,Y 453.035,Z 549.477,A -85,B 0,C 180,E1 -8370.889,E2 -8370.889} C_VEL
LIN {X 0,Y 452.867,Z 547.877,A -85,B 0,C 180,E1 -8372.668,E2 -8372.668} C_VEL
LIN {X 0,Y 452.878,Z 546.446,A -85,B 0,C 180,E1 -8373.559,E2 -8373.559} C_VEL
LIN {X 0,Y 452.851,Z 543.445,A -85,B 0,C 180,E1 -8374.896,E2 -8374.896} C_VEL
LIN {X 0,Y 452.843,Z 539.355,A -85,B 0,C 180,E1 -8376.237,E2 -8376.237} C_VEL
LIN {X 0,Y 452.89,Z 533.051,A -85,B 0,C 180,E1 -8377.804,E2 -8377.804} C_VEL
LIN {X 0,Y 453.013,Z 526.186,A -85,B 0,C 180,E1 -8379.15,E2 -8379.15} C_VEL
LIN {X 0,Y 453.302,Z 517.644,A -85,B 0,C 180,E1 -8380.496,E2 -8380.496} C_VEL
LIN {X 0,Y 453.639,Z 508.888,A -85,B 0,C 180,E1 -8381.619,E2 -8381.619} C_VEL
LIN {X 0,Y 454.162,Z 499.453,A -85,B 0,C 180,E1 -8382.616,E2 -8382.616} C_VEL
LIN {X 0,Y 454.644,Z 489.014,A -85,B 0,C 180,E1 -8383.521,E2 -8383.521} C_VEL
LIN {X 0,Y 455.192,Z 477.759,A -85,B 0,C 180,E1 -8384.302,E2 -8384.302} C_VEL
LIN {X 0,Y 455.656,Z 466.345,A -85,B 0,C 180,E1 -8384.915,E2 -8384.915} C_VEL
LIN {X 0,Y 454.634,Z 454.65,A -85,B 0,C 180,E1 -8385.423,E2 -8385.423} C_VEL
LIN {X 0,Y 453.108,Z 439.203,A -85,B 0,C 180,E1 -8385.916,E2 -8385.916} C_VEL
LIN {X 0,Y 453.324,Z 429.803,A -85,B 0,C 180,E1 -8388.063,E2 -8388.063} C_VEL
LIN {X 0,Y 453.666,Z 416.247,A -85,B 0,C 180,E1 -8391.271,E2 -8391.271} C_VEL
LIN {X 0,Y 454.116,Z 403.543,A -85,B 0,C 180,E1 -8394.326,E2 -8394.326} C_VEL
LIN {X 0,Y 454.617,Z 391.078,A -85,B 0,C 180,E1 -8397.381,E2 -8397.381} C_VEL
LIN {X 0,Y 455.22,Z 378.099,A -85,B 0,C 180,E1 -8400.628,E2 -8400.628} C_VEL
LIN {X 0,Y 455.992,Z 364.133,A -85,B 0,C 180,E1 -8404.232,E2 -8404.232} C_VEL
LIN {X 0,Y 456.63,Z 356.309,A -85,B 0,C 180,E1 -8406.297,E2 -8406.297} C_VEL
LIN {X 0,Y 456.093,Z 352.083,A -85,B 0,C 180,E1 -8407.492,E2 -8407.492} C_VEL
LIN {X 0,Y 454.008,Z 341.762,A -85,B 0,C 180,E1 -8410.552,E2 -8410.552} C_VEL
LIN {X 0,Y 453.502,Z 339.076,A -85,B 0,C 180,E1 -8411.415,E2 -8411.415} C_VEL
LIN {X 0,Y 453.476,Z 338.998,A -85,B 0,C 180,E1 -8414.528,E2 -8414.528} C_VEL
LIN {X 0,Y 453.44,Z 338.999,A -85,B 0,C 180,E1 -8418.069,E2 -8418.069} C_VEL
LIN {X 0,Y 453.441,Z 339,A -85,B 0,C 180,E1 -8420.8,E2 -8420.8} C_VEL
LIN {X 0,Y 453.446,Z 338.998,A -85,B 0,C 180,E1 -8423.916,E2 -8423.916} C_VEL
LIN {X 0,Y 453.471,Z 339.001,A -85,B 0,C 180,E1 -8427.15,E2 -8427.15} C_VEL
LIN {X 0,Y 453.465,Z 338.995,A -85,B 0,C 180,E1 -8430.267,E2 -8430.267} C_VEL
LIN {X 0,Y 453.494,Z 338.998,A -85,B 0,C 180,E1 -8433.293,E2 -8433.293} C_VEL
LIN {X 0,Y 453.487,Z 338.992,A -85,B 0,C 180,E1 -8436.238,E2 -8436.238} C_VEL
LIN {X 0,Y 453.473,Z 339.002,A -85,B 0,C 180,E1 -8439.117,E2 -8439.117} C_VEL
LIN {X 0,Y 453.493,Z 338.991,A -85,B 0,C 180,E1 -8441.944,E2 -8441.944} C_VEL
LIN {X 0,Y 453.529,Z 338.991,A -85,B 0,C 180,E1 -8444.726,E2 -8444.726} C_VEL
LIN {X 0,Y 453.549,Z 338.986,A -85,B 0,C 180,E1 -8448.379,E2 -8448.379} C_VEL
LIN {X 0,Y 453.575,Z 338.987,A -85,B 0,C 180,E1 -8451.086,E2 -8451.086} C_VEL
LIN {X 0,Y 453.655,Z 338.971,A -85,B 0,C 180,E1 -8453.774,E2 -8453.774} C_VEL
LIN {X 0,Y 453.732,Z 338.964,A -85,B 0,C 180,E1 -8457.337,E2 -8457.337} C_VEL
LIN {X 0,Y 453.811,Z 338.952,A -85,B 0,C 180,E1 -8460,E2 -8460} C_VEL
LIN {X 0,Y 453.732,Z 338.968,A -85,B 0,C 180,E1 -8462.663,E2 -8462.663} C_VEL
LIN {X 0,Y 453.658,Z 338.973,A -85,B 0,C 180,E1 -8466.226,E2 -8466.226} C_VEL
LIN {X 0,Y 453.582,Z 338.985,A -85,B 0,C 180,E1 -8468.914,E2 -8468.914} C_VEL
LIN {X 0,Y 453.554,Z 338.991,A -85,B 0,C 180,E1 -8472.529,E2 -8472.529} C_VEL
LIN {X 0,Y 453.535,Z 338.989,A -85,B 0,C 180,E1 -8476.196,E2 -8476.196} C_VEL
LIN {X 0,Y 453.511,Z 338.991,A -85,B 0,C 180,E1 -8479.041,E2 -8479.041} C_VEL
LIN {X 0,Y 453.47,Z 338.995,A -85,B 0,C 180,E1 -8481.836,E2 -8481.836} C_VEL
LIN {X 0,Y 453.507,Z 338.994,A -85,B 0,C 180,E1 -8484.735,E2 -8484.735} C_VEL
LIN {X 0,Y 453.525,Z 338.99,A -85,B 0,C 180,E1 -8487.961,E2 -8487.961} C_VEL
LIN {X 0,Y 453.476,Z 338.997,A -85,B 0,C 180,E1 -8490.76,E2 -8490.76} C_VEL
LIN {X 0,Y 453.471,Z 338.997,A -85,B 0,C 180,E1 -8493.913,E2 -8493.913} C_VEL
LIN {X 0,Y 453.464,Z 338.995,A -85,B 0,C 180,E1 -8497.189,E2 -8497.189} C_VEL
LIN {X 0,Y 453.521,Z 338.988,A -85,B 0,C 180,E1 -8499.447,E2 -8499.447} C_VEL
LIN {X 0,Y 453.473,Z 338.998,A -85,B 0,C 180,E1 -8501.936,E2 -8501.936} C_VEL
LIN {X 0,Y 453.487,Z 338.993,A -85,B 0,C 180,E1 -8505.471,E2 -8505.471} C_VEL
LIN {X 0,Y 453.478,Z 339,A -85,B 0,C 180,E1 -8508.21,E2 -8508.21} C_VEL
LIN {X 0,Y 453.512,Z 338.99,A -85,B 0,C 180,E1 -8510.791,E2 -8510.791} C_VEL
LIN {X 0,Y 453.454,Z 339.003,A -85,B 0,C 180,E1 -8513.918,E2 -8513.918} C_VEL
LIN {X 0,Y 453.481,Z 338.993,A -85,B 0,C 180,E1 -8517.152,E2 -8517.152} C_VEL
LIN {X 0,Y 453.513,Z 338.993,A -85,B 0,C 180,E1 -8520.272,E2 -8520.272} C_VEL
LIN {X 0,Y 453.514,Z 338.99,A -85,B 0,C 180,E1 -8523.295,E2 -8523.295} C_VEL
LIN {X 0,Y 453.505,Z 338.993,A -85,B 0,C 180,E1 -8526.24,E2 -8526.24} C_VEL
LIN {X 0,Y 453.484,Z 338.993,A -85,B 0,C 180,E1 -8529.118,E2 -8529.118} C_VEL
LIN {X 0,Y 453.514,Z 338.995,A -85,B 0,C 180,E1 -8531.945,E2 -8531.945} C_VEL
LIN {X 0,Y 453.552,Z 338.984,A -85,B 0,C 180,E1 -8534.727,E2 -8534.727} C_VEL
LIN {X 0,Y 453.562,Z 338.984,A -85,B 0,C 180,E1 -8538.379,E2 -8538.379} C_VEL
LIN {X 0,Y 453.655,Z 338.975,A -85,B 0,C 180,E1 -8541.985,E2 -8541.985} C_VEL
LIN {X 0,Y 453.641,Z 338.974,A -85,B 0,C 180,E1 -8543.108,E2 -8543.108} C_VEL
LIN {X 0,Y 452.957,Z 339.063,A -85,B 0,C 180,E1 -8543.848,E2 -8543.848} C_VEL
LIN {X 0,Y 450.008,Z 339.427,A -85,B 0,C 180,E1 -8545.05,E2 -8545.05} C_VEL
LIN {X 0,Y 447.585,Z 339.73,A -85,B 0,C 180,E1 -8546.019,E2 -8546.019} C_VEL
LIN {X 0,Y 446.65,Z 339.845,A -85,B 0,C 180,E1 -8546.769,E2 -8546.769} C_VEL
LIN {X 0,Y 446.63,Z 339.848,A -85,B 0,C 180,E1 -8547.023,E2 -8547.023} C_VEL
LIN {X 0,Y 446.797,Z 339.828,A -85,B 0,C 180,E1 -8550,E2 -8550} C_VEL
LIN {X 0,Y 446.712,Z 339.836,A -85,B 0,C 180,E1 -8552.705,E2 -8552.705} C_VEL
LIN {X 0,Y 446.642,Z 339.845,A -85,B 0,C 180,E1 -8556.324,E2 -8556.324} C_VEL
LIN {X 0,Y 446.54,Z 339.861,A -85,B 0,C 180,E1 -8559.055,E2 -8559.055} C_VEL
LIN {X 0,Y 446.523,Z 339.861,A -85,B 0,C 180,E1 -8562.729,E2 -8562.729} C_VEL
LIN {X 0,Y 446.498,Z 339.863,A -85,B 0,C 180,E1 -8566.228,E2 -8566.228} C_VEL
LIN {X 0,Y 446.471,Z 339.874,A -85,B 0,C 180,E1 -8569.303,E2 -8569.303} C_VEL
LIN {X 0,Y 446.419,Z 339.873,A -85,B 0,C 180,E1 -8572.199,E2 -8572.199} C_VEL
LIN {X 0,Y 446.459,Z 339.875,A -85,B 0,C 180,E1 -8575.152,E2 -8575.152} C_VEL
LIN {X 0,Y 446.484,Z 339.865,A -85,B 0,C 180,E1 -8578.178,E2 -8578.178} C_VEL
LIN {X 0,Y 446.419,Z 339.874,A -85,B 0,C 180,E1 -8581.774,E2 -8581.774} C_VEL
LIN {X 0,Y 446.429,Z 339.873,A -85,B 0,C 180,E1 -8584.522,E2 -8584.522} C_VEL
LIN {X 0,Y 446.437,Z 339.87,A -85,B 0,C 180,E1 -8588.082,E2 -8588.082} C_VEL
LIN {X 0,Y 446.445,Z 339.877,A -85,B 0,C 180,E1 -8590.92,E2 -8590.92} C_VEL
LIN {X 0,Y 446.441,Z 339.874,A -85,B 0,C 180,E1 -8593.84,E2 -8593.84} C_VEL
LIN {X 0,Y 446.519,Z 340.061,A -85,B 0,C 180,E1 -8596.796,E2 -8596.796} C_VEL
LIN {X 0,Y 446.818,Z 341.306,A -85,B 0,C 180,E1 -8596.961,E2 -8596.961} C_VEL
LIN {X 0,Y 449.436,Z 350.476,A -85,B 0,C 180,E1 -8597.588,E2 -8597.588} C_VEL
LIN {X 0,Y 449.325,Z 360.324,A -85,B 0,C 180,E1 -8598.28,E2 -8598.28} C_VEL
LIN {X 0,Y 448.816,Z 370.775,A -85,B 0,C 180,E1 -8599.174,E2 -8599.174} C_VEL
LIN {X 0,Y 448.362,Z 380.291,A -85,B 0,C 180,E1 -8600.179,E2 -8600.179} C_VEL
LIN {X 0,Y 447.809,Z 390.211,A -85,B 0,C 180,E1 -8601.465,E2 -8601.465} C_VEL
LIN {X 0,Y 447.381,Z 398.382,A -85,B 0,C 180,E1 -8602.786,E2 -8602.786} C_VEL
LIN {X 0,Y 447.013,Z 405.178,A -85,B 0,C 180,E1 -8604.151,E2 -8604.151} C_VEL
LIN {X 0,Y 446.701,Z 410.569,A -85,B 0,C 180,E1 -8605.501,E2 -8605.501} C_VEL
LIN {X 0,Y 446.462,Z 415.505,A -85,B 0,C 180,E1 -8607.106,E2 -8607.106} C_VEL
LIN {X 0,Y 446.321,Z 418.911,A -85,B 0,C 180,E1 -8608.692,E2 -8608.692} C_VEL
LIN {X 0,Y 446.228,Z 420.8,A -85,B 0,C 180,E1 -8610.022,E2 -8610.022} C_VEL
LIN {X 0,Y 446.164,Z 421.947,A -85,B 0,C 180,E1 -8611.799,E2 -8611.799} C_VEL
LIN {X 0,Y 446.18,Z 421.942,A -85,B 0,C 180,E1 -8612.82,E2 -8612.82} C_VEL
LIN {X 0,Y 446.245,Z 421.377,A -85,B 0,C 180,E1 -8613.855,E2 -8613.855} C_VEL
LIN {X 0,Y 446.36,Z 420.393,A -85,B 0,C 180,E1 -8614.842,E2 -8614.842} C_VEL
LIN {X 0,Y 446.459,Z 418.721,A -85,B 0,C 180,E1 -8615.922,E2 -8615.922} C_VEL
LIN {X 0,Y 446.712,Z 415.653,A -85,B 0,C 180,E1 -8617.328,E2 -8617.328} C_VEL
LIN {X 0,Y 446.977,Z 411.262,A -85,B 0,C 180,E1 -8618.799,E2 -8618.799} C_VEL
LIN {X 0,Y 447.359,Z 405.841,A -85,B 0,C 180,E1 -8620.192,E2 -8620.192} C_VEL
LIN {X 0,Y 447.778,Z 399.606,A -85,B 0,C 180,E1 -8621.468,E2 -8621.468} C_VEL
LIN {X 0,Y 448.28,Z 391.362,A -85,B 0,C 180,E1 -8622.822,E2 -8622.822} C_VEL
LIN {X 0,Y 448.852,Z 381.711,A -85,B 0,C 180,E1 -8624.097,E2 -8624.097} C_VEL
LIN {X 0,Y 449.429,Z 371.56,A -85,B 0,C 180,E1 -8625.163,E2 -8625.163} C_VEL
LIN {X 0,Y 449.865,Z 360.895,A -85,B 0,C 180,E1 -8626.068,E2 -8626.068} C_VEL
LIN {X 0,Y 450.068,Z 352.002,A -85,B 0,C 180,E1 -8626.684,E2 -8626.684} C_VEL
LIN {X 0,Y 446.695,Z 340.601,A -85,B 0,C 180,E1 -8627.504,E2 -8627.504} C_VEL
LIN {X 0,Y 446.548,Z 339.895,A -85,B 0,C 180,E1 -8627.698,E2 -8627.698} C_VEL
LIN {X 0,Y 446.529,Z 339.865,A -85,B 0,C 180,E1 -8630.944,E2 -8630.944} C_VEL
LIN {X 0,Y 446.627,Z 339.853,A -85,B 0,C 180,E1 -8633.676,E2 -8633.676} C_VEL
LIN {X 0,Y 446.679,Z 339.846,A -85,B 0,C 180,E1 -8637.295,E2 -8637.295} C_VEL
LIN {X 0,Y 446.781,Z 339.831,A -85,B 0,C 180,E1 -8640,E2 -8640} C_VEL
LIN {X 0,Y 446.679,Z 339.844,A -85,B 0,C 180,E1 -8642.706,E2 -8642.706} C_VEL
LIN {X 0,Y 446.623,Z 339.849,A -85,B 0,C 180,E1 -8646.324,E2 -8646.324} C_VEL
LIN {X 0,Y 446.522,Z 339.866,A -85,B 0,C 180,E1 -8649.056,E2 -8649.056} C_VEL
LIN {X 0,Y 446.512,Z 339.865,A -85,B 0,C 180,E1 -8652.73,E2 -8652.73} C_VEL
LIN {X 0,Y 446.486,Z 339.866,A -85,B 0,C 180,E1 -8656.228,E2 -8656.228} C_VEL
LIN {X 0,Y 446.459,Z 339.873,A -85,B 0,C 180,E1 -8659.304,E2 -8659.304} C_VEL
LIN {X 0,Y 446.408,Z 339.876,A -85,B 0,C 180,E1 -8662.2,E2 -8662.2} C_VEL
LIN {X 0,Y 446.438,Z 339.876,A -85,B 0,C 180,E1 -8665.154,E2 -8665.154} C_VEL
LIN {X 0,Y 446.477,Z 339.868,A -85,B 0,C 180,E1 -8668.179,E2 -8668.179} C_VEL
LIN {X 0,Y 446.41,Z 339.876,A -85,B 0,C 180,E1 -8671.775,E2 -8671.775} C_VEL
LIN {X 0,Y 446.415,Z 339.879,A -85,B 0,C 180,E1 -8674.524,E2 -8674.524} C_VEL
LIN {X 0,Y 446.405,Z 339.879,A -85,B 0,C 180,E1 -8678.079,E2 -8678.079} C_VEL
LIN {X 0,Y 446.396,Z 339.88,A -85,B 0,C 180,E1 -8681.395,E2 -8681.395} C_VEL
LIN {X 0,Y 446.444,Z 339.876,A -85,B 0,C 180,E1 -8685.105,E2 -8685.105} C_VEL
LIN {X 0,Y 446.407,Z 339.882,A -85,B 0,C 180,E1 -8688.608,E2 -8688.608} C_VEL
LIN {X 0,Y 446.455,Z 340.106,A -85,B 0,C 180,E1 -8689.161,E2 -8689.161} C_VEL
LIN {X 0,Y 448.373,Z 349.668,A -85,B 0,C 180,E1 -8692.317,E2 -8692.317} C_VEL
LIN {X 0,Y 448.907,Z 353.542,A -85,B 0,C 180,E1 -8693.494,E2 -8693.494} C_VEL
LIN {X 0,Y 448.504,Z 359.312,A -85,B 0,C 180,E1 -8695.115,E2 -8695.115} C_VEL
LIN {X 0,Y 447.745,Z 373.092,A -85,B 0,C 180,E1 -8698.804,E2 -8698.804} C_VEL
LIN {X 0,Y 447.158,Z 387.124,A -85,B 0,C 180,E1 -8702.378,E2 -8702.378} C_VEL
LIN {X 0,Y 446.733,Z 400.327,A -85,B 0,C 180,E1 -8705.609,E2 -8705.609} C_VEL
LIN {X 0,Y 446.38,Z 415.615,A -85,B 0,C 180,E1 -8709.253,E2 -8709.253} C_VEL
LIN {X 0,Y 446.14,Z 429.871,A -85,B 0,C 180,E1 -8712.585,E2 -8712.585} C_VEL
LIN {X 0,Y 446.039,Z 435.069,A -85,B 0,C 180,E1 -8713.719,E2 -8713.719} C_VEL
LIN {X 0,Y 447.6,Z 452.489,A -85,B 0,C 180,E1 -8714.308,E2 -8714.308} C_VEL
LIN {X 0,Y 448.258,Z 464.031,A -85,B 0,C 180,E1 -8714.833,E2 -8714.833} C_VEL
LIN {X 0,Y 448.503,Z 469.512,A -85,B 0,C 180,E1 -8715.132,E2 -8715.132} C_VEL
LIN {X 0,Y 447.847,Z 481.94,A -85,B 0,C 180,E1 -8715.923,E2 -8715.923} C_VEL
LIN {X 0,Y 447.288,Z 493.315,A -85,B 0,C 180,E1 -8716.839,E2 -8716.839} C_VEL
LIN {X 0,Y 446.898,Z 503.545,A -85,B 0,C 180,E1 -8717.858,E2 -8717.858} C_VEL
LIN {X 0,Y 446.437,Z 512.059,A -85,B 0,C 180,E1 -8718.881,E2 -8718.881} C_VEL
LIN {X 0,Y 446.026,Z 521.387,A -85,B 0,C 180,E1 -8720.248,E2 -8720.248} C_VEL
LIN {X 0,Y 445.858,Z 528.974,A -85,B 0,C 180,E1 -8721.616,E2 -8721.616} C_VEL
LIN {X 0,Y 445.793,Z 535.311,A -85,B 0,C 180,E1 -8723.04,E2 -8723.04} C_VEL
LIN {X 0,Y 445.796,Z 540.582,A -85,B 0,C 180,E1 -8724.572,E2 -8724.572} C_VEL
LIN {X 0,Y 445.857,Z 544.1,A -85,B 0,C 180,E1 -8725.933,E2 -8725.933} C_VEL
LIN {X 0,Y 445.854,Z 546.579,A -85,B 0,C 180,E1 -8727.29,E2 -8727.29} C_VEL
LIN {X 0,Y 446.016,Z 548.392,A -85,B 0,C 180,E1 -8729.097,E2 -8729.097} C_VEL
LIN {X 0,Y 446.009,Z 548.662,A -85,B 0,C 180,E1 -8730,E2 -8730} C_VEL
LIN {X 0,Y 446.012,Z 548.482,A -85,B 0,C 180,E1 -8730.903,E2 -8730.903} C_VEL
LIN {X 0,Y 445.823,Z 546.882,A -85,B 0,C 180,E1 -8732.711,E2 -8732.711} C_VEL
LIN {X 0,Y 445.836,Z 545.446,A -85,B 0,C 180,E1 -8733.615,E2 -8733.615} C_VEL
LIN {X 0,Y 445.802,Z 542.44,A -85,B 0,C 180,E1 -8734.974,E2 -8734.974} C_VEL
LIN {X 0,Y 445.771,Z 537.187,A -85,B 0,C 180,E1 -8736.657,E2 -8736.657} C_VEL
LIN {X 0,Y 445.851,Z 531.012,A -85,B 0,C 180,E1 -8738.156,E2 -8738.156} C_VEL
LIN {X 0,Y 445.979,Z 523.846,A -85,B 0,C 180,E1 -8739.524,E2 -8739.524} C_VEL
LIN {X 0,Y 446.356,Z 514.955,A -85,B 0,C 180,E1 -8740.891,E2 -8740.891} C_VEL
LIN {X 0,Y 446.796,Z 505.872,A -85,B 0,C 180,E1 -8742.029,E2 -8742.029} C_VEL
LIN {X 0,Y 447.304,Z 495.288,A -85,B 0,C 180,E1 -8743.106,E2 -8743.106} C_VEL
LIN {X 0,Y 447.915,Z 483.326,A -85,B 0,C 180,E1 -8744.075,E2 -8744.075} C_VEL
LIN {X 0,Y 448.525,Z 471.742,A -85,B 0,C 180,E1 -8744.809,E2 -8744.809} C_VEL
LIN {X 0,Y 448.59,Z 466.273,A -85,B 0,C 180,E1 -8745.097,E2 -8745.097} C_VEL
LIN {X 0,Y 447.658,Z 454.52,A -85,B 0,C 180,E1 -8745.625,E2 -8745.625} C_VEL
LIN {X 0,Y 446.038,Z 438.124,A -85,B 0,C 180,E1 -8746.177,E2 -8746.177} C_VEL
LIN {X 0,Y 446.38,Z 424.92,A -85,B 0,C 180,E1 -8749.307,E2 -8749.307} C_VEL
LIN {X 0,Y 446.817,Z 411.08,A -85,B 0,C 180,E1 -8752.666,E2 -8752.666} C_VEL
LIN {X 0,Y 447.361,Z 397.195,A -85,B 0,C 180,E1 -8756.095,E2 -8756.095} C_VEL
LIN {X 0,Y 447.836,Z 385.277,A -85,B 0,C 180,E1 -8759.109,E2 -8759.109} C_VEL
LIN {X 0,Y 448.391,Z 375.319,A -85,B 0,C 180,E1 -8761.672,E2 -8761.672} C_VEL
LIN {X 0,Y 449.368,Z 361.395,A -85,B 0,C 180,E1 -8765.356,E2 -8765.356} C_VEL
LIN {X 0,Y 449.599,Z 356.212,A -85,B 0,C 180,E1 -8766.765,E2 -8766.765} C_VEL
LIN {X 0,Y 447.697,Z 346.281,A -85,B 0,C 180,E1 -8769.717,E2 -8769.717} C_VEL
LIN {X 0,Y 446.422,Z 339.972,A -85,B 0,C 180,E1 -8771.692,E2 -8771.692} C_VEL
LIN {X 0,Y 446.444,Z 339.876,A -85,B 0,C 180,E1 -8775.103,E2 -8775.103} C_VEL
LIN {X 0,Y 446.399,Z 339.876,A -85,B 0,C 180,E1 -8778.605,E2 -8778.605} C_VEL
LIN {X 0,Y 446.405,Z 339.876,A -85,B 0,C 180,E1 -8781.921,E2 -8781.921} C_VEL
LIN {X 0,Y 446.415,Z 339.878,A -85,B 0,C 180,E1 -8785.476,E2 -8785.476} C_VEL
LIN {X 0,Y 446.407,Z 339.876,A -85,B 0,C 180,E1 -8788.699,E2 -8788.699} C_VEL
LIN {X 0,Y 446.477,Z 339.867,A -85,B 0,C 180,E1 -8791.821,E2 -8791.821} C_VEL
LIN {X 0,Y 446.435,Z 339.875,A -85,B 0,C 180,E1 -8794.846,E2 -8794.846} C_VEL
LIN {X 0,Y 446.439,Z 339.87,A -85,B 0,C 180,E1 -8798.245,E2 -8798.245} C_VEL
LIN {X 0,Y 446.442,Z 339.871,A -85,B 0,C 180,E1 -8801.648,E2 -8801.648} C_VEL
LIN {X 0,Y 446.498,Z 339.865,A -85,B 0,C 180,E1 -8804.479,E2 -8804.479} C_VEL
LIN {X 0,Y 446.507,Z 339.862,A -85,B 0,C 180,E1 -8808.193,E2 -8808.193} C_VEL
LIN {X 0,Y 446.522,Z 339.868,A -85,B 0,C 180,E1 -8810.944,E2 -8810.944} C_VEL
LIN {X 0,Y 446.623,Z 339.848,A -85,B 0,C 180,E1 -8813.676,E2 -8813.676} C_VEL
LIN {X 0,Y 446.679,Z 339.843,A -85,B 0,C 180,E1 -8817.294,E2 -8817.294} C_VEL
LIN {X 0,Y 446.781,Z 339.828,A -85,B 0,C 180,E1 -8820,E2 -8820} C_VEL
LIN {X 0,Y 446.679,Z 339.848,A -85,B 0,C 180,E1 -8822.705,E2 -8822.705} C_VEL
LIN {X 0,Y 446.627,Z 339.85,A -85,B 0,C 180,E1 -8826.324,E2 -8826.324} C_VEL
LIN {X 0,Y 446.528,Z 339.862,A -85,B 0,C 180,E1 -8829.056,E2 -8829.056} C_VEL
LIN {X 0,Y 446.512,Z 339.868,A -85,B 0,C 180,E1 -8832.73,E2 -8832.73} C_VEL
LIN {X 0,Y 446.487,Z 339.868,A -85,B 0,C 180,E1 -8836.228,E2 -8836.228} C_VEL
LIN {X 0,Y 446.46,Z 339.868,A -85,B 0,C 180,E1 -8839.304,E2 -8839.304} C_VEL
LIN {X 0,Y 446.413,Z 339.878,A -85,B 0,C 180,E1 -8842.2,E2 -8842.2} C_VEL
LIN {X 0,Y 446.45,Z 339.87,A -85,B 0,C 180,E1 -8845.153,E2 -8845.153} C_VEL
LIN {X 0,Y 446.477,Z 339.87,A -85,B 0,C 180,E1 -8848.179,E2 -8848.179} C_VEL
LIN {X 0,Y 446.412,Z 339.874,A -85,B 0,C 180,E1 -8851.301,E2 -8851.301} C_VEL
LIN {X 0,Y 446.424,Z 339.877,A -85,B 0,C 180,E1 -8854.524,E2 -8854.524} C_VEL
LIN {X 0,Y 446.428,Z 339.877,A -85,B 0,C 180,E1 -8858.083,E2 -8858.083} C_VEL
LIN {X 0,Y 446.438,Z 339.871,A -85,B 0,C 180,E1 -8860.921,E2 -8860.921} C_VEL
LIN {X 0,Y 446.396,Z 339.879,A -85,B 0,C 180,E1 -8863.847,E2 -8863.847} C_VEL
LIN {X 0,Y 446.416,Z 339.878,A -85,B 0,C 180,E1 -8866.401,E2 -8866.401} C_VEL
LIN {X 0,Y 446.448,Z 339.873,A -85,B 0,C 180,E1 -8869.804,E2 -8869.804} C_VEL
LIN {X 0,Y 446.425,Z 339.879,A -85,B 0,C 180,E1 -8872.124,E2 -8872.124} C_VEL
LIN {X 0,Y 446.428,Z 339.873,A -85,B 0,C 180,E1 -8875.478,E2 -8875.478} C_VEL
LIN {X 0,Y 446.418,Z 339.873,A -85,B 0,C 180,E1 -8878.701,E2 -8878.701} C_VEL
LIN {X 0,Y 446.484,Z 339.871,A -85,B 0,C 180,E1 -8881.822,E2 -8881.822} C_VEL
LIN {X 0,Y 446.459,Z 339.868,A -85,B 0,C 180,E1 -8884.848,E2 -8884.848} C_VEL
LIN {X 0,Y 446.449,Z 339.872,A -85,B 0,C 180,E1 -8888.245,E2 -8888.245} C_VEL
LIN {X 0,Y 446.46,Z 339.874,A -85,B 0,C 180,E1 -8891.65,E2 -8891.65} C_VEL
LIN {X 0,Y 446.518,Z 339.861,A -85,B 0,C 180,E1 -8894.481,E2 -8894.481} C_VEL
LIN {X 0,Y 446.52,Z 339.862,A -85,B 0,C 180,E1 -8898.193,E2 -8898.193} C_VEL
LIN {X 0,Y 446.603,Z 339.855,A -85,B 0,C 180,E1 -8901.858,E2 -8901.858} C_VEL
LIN {X 0,Y 446.65,Z 339.844,A -85,B 0,C 180,E1 -8904.583,E2 -8904.583} C_VEL
LIN {X 0,Y 446.63,Z 339.848,A -85,B 0,C 180,E1 -8907.023,E2 -8907.023} C_VEL
LIN {X 0,Y 446.114,Z 339.918,A -85,B 0,C 180,E1 -8907.776,E2 -8907.776} C_VEL
LIN {X 0,Y 443.295,Z 340.269,A -85,B 0,C 180,E1 -8908.999,E2 -8908.999} C_VEL
LIN {X 0,Y 440.807,Z 340.576,A -85,B 0,C 180,E1 -8909.986,E2 -8909.986} C_VEL
LIN {X 0,Y 439.718,Z 340.709,A -85,B 0,C 180,E1 -8910.749,E2 -8910.749} C_VEL
LIN {X 0,Y 439.624,Z 340.72,A -85,B 0,C 180,E1 -8911.008,E2 -8911.008} C_VEL
LIN {X 0,Y 439.659,Z 340.715,A -85,B 0,C 180,E1 -8912.749,E2 -8912.749} C_VEL
LIN {X 0,Y 439.614,Z 340.72,A -85,B 0,C 180,E1 -8916.425,E2 -8916.425} C_VEL
LIN {X 0,Y 439.502,Z 340.739,A -85,B 0,C 180,E1 -8919.201,E2 -8919.201} C_VEL
LIN {X 0,Y 439.468,Z 340.741,A -85,B 0,C 180,E1 -8922.937,E2 -8922.937} C_VEL
LIN {X 0,Y 439.449,Z 340.741,A -85,B 0,C 180,E1 -8926.348,E2 -8926.348} C_VEL
LIN {X 0,Y 439.404,Z 340.75,A -85,B 0,C 180,E1 -8929.626,E2 -8929.626} C_VEL
LIN {X 0,Y 439.366,Z 340.752,A -85,B 0,C 180,E1 -8932.575,E2 -8932.575} C_VEL
LIN {X 0,Y 439.406,Z 340.749,A -85,B 0,C 180,E1 -8935.584,E2 -8935.584} C_VEL
LIN {X 0,Y 439.417,Z 340.747,A -85,B 0,C 180,E1 -8938.673,E2 -8938.673} C_VEL
LIN {X 0,Y 439.369,Z 340.751,A -85,B 0,C 180,E1 -8942.03,E2 -8942.03} C_VEL
LIN {X 0,Y 439.395,Z 340.752,A -85,B 0,C 180,E1 -8945.34,E2 -8945.34} C_VEL
LIN {X 0,Y 439.397,Z 340.75,A -85,B 0,C 180,E1 -8948.592,E2 -8948.592} C_VEL
LIN {X 0,Y 439.402,Z 340.754,A -85,B 0,C 180,E1 -8951.259,E2 -8951.259} C_VEL
LIN {X 0,Y 439.406,Z 340.753,A -85,B 0,C 180,E1 -8954.727,E2 -8954.727} C_VEL
LIN {X 0,Y 439.46,Z 340.905,A -85,B 0,C 180,E1 -8956.554,E2 -8956.554} C_VEL
LIN {X 0,Y 439.755,Z 342.122,A -85,B 0,C 180,E1 -8956.729,E2 -8956.729} C_VEL
LIN {X 0,Y 442.673,Z 352.59,A -85,B 0,C 180,E1 -8957.464,E2 -8957.464} C_VEL
LIN {X 0,Y 442.309,Z 364.041,A -85,B 0,C 180,E1 -8958.312,E2 -8958.312} C_VEL
LIN {X 0,Y 441.788,Z 374.659,A -85,B 0,C 180,E1 -8959.29,E2 -8959.29} C_VEL
LIN {X 0,Y 441.274,Z 384.62,A -85,B 0,C 180,E1 -8960.427,E2 -8960.427} C_VEL
LIN {X 0,Y 440.772,Z 392.681,A -85,B 0,C 180,E1 -8961.549,E2 -8961.549} C_VEL
LIN {X 0,Y 440.324,Z 400.84,A -85,B 0,C 180,E1 -8962.942,E2 -8962.942} C_VEL
LIN {X 0,Y 440.006,Z 406.898,A -85,B 0,C 180,E1 -8964.22,E2 -8964.22} C_VEL
LIN {X 0,Y 439.697,Z 411.586,A -85,B 0,C 180,E1 -8965.429,E2 -8965.429} C_VEL
LIN {X 0,Y 439.468,Z 416.524,A -85,B 0,C 180,E1 -8967.062,E2 -8967.062} C_VEL
LIN {X 0,Y 439.372,Z 418.933,A -85,B 0,C 180,E1 -8968.139,E2 -8968.139} C_VEL
LIN {X 0,Y 439.21,Z 421.537,A -85,B 0,C 180,E1 -8969.775,E2 -8969.775} C_VEL
LIN {X 0,Y 439.154,Z 422.915,A -85,B 0,C 180,E1 -8971.663,E2 -8971.663} C_VEL
LIN {X 0,Y 439.185,Z 422.745,A -85,B 0,C 180,E1 -8973.38,E2 -8973.38} C_VEL
LIN {X 0,Y 439.285,Z 421.968,A -85,B 0,C 180,E1 -8974.408,E2 -8974.408} C_VEL
LIN {X 0,Y 439.447,Z 420.257,A -85,B 0,C 180,E1 -8975.723,E2 -8975.723} C_VEL
LIN {X 0,Y 439.734,Z 416.663,A -85,B 0,C 180,E1 -8977.445,E2 -8977.445} C_VEL
LIN {X 0,Y 440.052,Z 412.258,A -85,B 0,C 180,E1 -8978.94,E2 -8978.94} C_VEL
LIN {X 0,Y 440.45,Z 406.54,A -85,B 0,C 180,E1 -8980.422,E2 -8980.422} C_VEL
LIN {X 0,Y 440.967,Z 399.226,A -85,B 0,C 180,E1 -8981.893,E2 -8981.893} C_VEL
LIN {X 0,Y 441.494,Z 391.341,A -85,B 0,C 180,E1 -8983.17,E2 -8983.17} C_VEL
LIN {X 0,Y 442.05,Z 382.635,A -85,B 0,C 180,E1 -8984.319,E2 -8984.319} C_VEL
LIN {X 0,Y 442.657,Z 372.258,A -85,B 0,C 180,E1 -8985.42,E2 -8985.42} C_VEL
LIN {X 0,Y 443.132,Z 361.266,A -85,B 0,C 180,E1 -8986.359,E2 -8986.359} C_VEL
LIN {X 0,Y 443.432,Z 354.758,A -85,B 0,C 180,E1 -8986.818,E2 -8986.818} C_VEL
LIN {X 0,Y 441.432,Z 347.115,A -85,B 0,C 180,E1 -8987.385,E2 -8987.385} C_VEL
LIN {X 0,Y 439.646,Z 341.498,A -85,B 0,C 180,E1 -8987.796,E2 -8987.796} C_VEL
LIN {X 0,Y 439.511,Z 340.769,A -85,B 0,C 180,E1 -8988.002,E2 -8988.002} C_VEL
LIN {X 0,Y 439.538,Z 340.735,A -85,B 0,C 180,E1 -8991.726,E2 -8991.726} C_VEL
LIN {X 0,Y 439.605,Z 340.725,A -85,B 0,C 180,E1 -8994.496,E2 -8994.496} C_VEL
LIN {X 0,Y 439.622,Z 340.722,A -85,B 0,C 180,E1 -8998.168,E2 -8998.168} C_VEL
LIN {X 0,Y 439.751,Z 340.707,A -85,B 0,C 180,E1 -9000,E2 -9000} C_VEL
LIN {X 0,Y 439.629,Z 340.723,A -85,B 0,C 180,E1 -9002.749,E2 -9002.749} C_VEL
LIN {X 0,Y 439.594,Z 340.725,A -85,B 0,C 180,E1 -9006.426,E2 -9006.426} C_VEL
LIN {X 0,Y 439.485,Z 340.744,A -85,B 0,C 180,E1 -9009.202,E2 -9009.202} C_VEL
LIN {X 0,Y 439.456,Z 340.746,A -85,B 0,C 180,E1 -9012.938,E2 -9012.938} C_VEL
LIN {X 0,Y 439.437,Z 340.745,A -85,B 0,C 180,E1 -9016.348,E2 -9016.348} C_VEL
LIN {X 0,Y 439.393,Z 340.75,A -85,B 0,C 180,E1 -9019.627,E2 -9019.627} C_VEL
LIN {X 0,Y 439.355,Z 340.757,A -85,B 0,C 180,E1 -9022.576,E2 -9022.576} C_VEL
LIN {X 0,Y 439.39,Z 340.75,A -85,B 0,C 180,E1 -9025.586,E2 -9025.586} C_VEL
LIN {X 0,Y 439.409,Z 340.751,A -85,B 0,C 180,E1 -9028.674,E2 -9028.674} C_VEL
LIN {X 0,Y 439.36,Z 340.754,A -85,B 0,C 180,E1 -9032.031,E2 -9032.031} C_VEL
LIN {X 0,Y 439.385,Z 340.753,A -85,B 0,C 180,E1 -9035.341,E2 -9035.341} C_VEL
LIN {X 0,Y 439.356,Z 340.759,A -85,B 0,C 180,E1 -9038.598,E2 -9038.598} C_VEL
LIN {X 0,Y 439.345,Z 340.759,A -85,B 0,C 180,E1 -9042.211,E2 -9042.211} C_VEL
LIN {X 0,Y 439.392,Z 340.755,A -85,B 0,C 180,E1 -9045.271,E2 -9045.271} C_VEL
LIN {X 0,Y 439.378,Z 340.882,A -85,B 0,C 180,E1 -9048.745,E2 -9048.745} C_VEL
LIN {X 0,Y 441.061,Z 349.093,A -85,B 0,C 180,E1 -9051.58,E2 -9051.58} C_VEL
LIN {X 0,Y 441.97,Z 354.842,A -85,B 0,C 180,E1 -9053.395,E2 -9053.395} C_VEL
LIN {X 0,Y 441.563,Z 360.601,A -85,B 0,C 180,E1 -9055.043,E2 -9055.043} C_VEL
LIN {X 0,Y 440.737,Z 374.286,A -85,B 0,C 180,E1 -9058.786,E2 -9058.786} C_VEL
LIN {X 0,Y 440.139,Z 387.27,A -85,B 0,C 180,E1 -9062.157,E2 -9062.157} C_VEL
LIN {X 0,Y 439.687,Z 400.39,A -85,B 0,C 180,E1 -9065.444,E2 -9065.444} C_VEL
LIN {X 0,Y 439.308,Z 415.627,A -85,B 0,C 180,E1 -9069.149,E2 -9069.149} C_VEL
LIN {X 0,Y 439.058,Z 429.837,A -85,B 0,C 180,E1 -9072.535,E2 -9072.535} C_VEL
LIN {X 0,Y 438.947,Z 433.773,A -85,B 0,C 180,E1 -9073.413,E2 -9073.413} C_VEL
LIN {X 0,Y 439.167,Z 436.055,A -85,B 0,C 180,E1 -9073.52,E2 -9073.52} C_VEL
LIN {X 0,Y 440.46,Z 449.435,A -85,B 0,C 180,E1 -9073.958,E2 -9073.958} C_VEL
LIN {X 0,Y 441.141,Z 462.07,A -85,B 0,C 180,E1 -9074.523,E2 -9074.523} C_VEL
LIN {X 0,Y 441.616,Z 468.687,A -85,B 0,C 180,E1 -9074.895,E2 -9074.895} C_VEL
LIN {X 0,Y 440.933,Z 481.018,A -85,B 0,C 180,E1 -9075.697,E2 -9075.697} C_VEL
LIN {X 0,Y 440.293,Z 492.756,A -85,B 0,C 180,E1 -9076.665,E2 -9076.665} C_VEL
LIN {X 0,Y 439.843,Z 503.514,A -85,B 0,C 180,E1 -9077.777,E2 -9077.777} C_VEL
LIN {X 0,Y 439.322,Z 512.702,A -85,B 0,C 180,E1 -9078.933,E2 -9078.933} C_VEL
LIN {X 0,Y 438.947,Z 521.761,A -85,B 0,C 180,E1 -9080.322,E2 -9080.322} C_VEL
LIN {X 0,Y 438.778,Z 529.047,A -85,B 0,C 180,E1 -9081.712,E2 -9081.712} C_VEL
LIN {X 0,Y 438.712,Z 535.752,A -85,B 0,C 180,E1 -9083.325,E2 -9083.325} C_VEL
LIN {X 0,Y 438.791,Z 540.882,A -85,B 0,C 180,E1 -9084.946,E2 -9084.946} C_VEL
LIN {X 0,Y 438.818,Z 544.049,A -85,B 0,C 180,E1 -9086.327,E2 -9086.327} C_VEL
LIN {X 0,Y 438.811,Z 545.569,A -85,B 0,C 180,E1 -9087.246,E2 -9087.246} C_VEL
LIN {X 0,Y 438.993,Z 547.394,A -85,B 0,C 180,E1 -9089.083,E2 -9089.083} C_VEL
LIN {X 0,Y 438.989,Z 547.662,A -85,B 0,C 180,E1 -9090,E2 -9090} C_VEL
LIN {X 0,Y 438.989,Z 547.482,A -85,B 0,C 180,E1 -9090.917,E2 -9090.917} C_VEL
LIN {X 0,Y 438.78,Z 545.88,A -85,B 0,C 180,E1 -9092.754,E2 -9092.754} C_VEL
LIN {X 0,Y 438.794,Z 544.437,A -85,B 0,C 180,E1 -9093.673,E2 -9093.673} C_VEL
LIN {X 0,Y 438.752,Z 541.422,A -85,B 0,C 180,E1 -9095.054,E2 -9095.054} C_VEL
LIN {X 0,Y 438.727,Z 536.412,A -85,B 0,C 180,E1 -9096.693,E2 -9096.693} C_VEL
LIN {X 0,Y 438.77,Z 529.96,A -85,B 0,C 180,E1 -9098.288,E2 -9098.288} C_VEL
LIN {X 0,Y 438.915,Z 522.771,A -85,B 0,C 180,E1 -9099.679,E2 -9099.679} C_VEL
LIN {X 0,Y 439.319,Z 513.864,A -85,B 0,C 180,E1 -9101.067,E2 -9101.067} C_VEL
LIN {X 0,Y 439.843,Z 504.77,A -85,B 0,C 180,E1 -9102.223,E2 -9102.223} C_VEL
LIN {X 0,Y 440.342,Z 493.951,A -85,B 0,C 180,E1 -9103.334,E2 -9103.334} C_VEL
LIN {X 0,Y 440.872,Z 483.682,A -85,B 0,C 180,E1 -9104.187,E2 -9104.187} C_VEL
LIN {X 0,Y 441.578,Z 471.501,A -85,B 0,C 180,E1 -9104.988,E2 -9104.988} C_VEL
LIN {X 0,Y 441.498,Z 466.115,A -85,B 0,C 180,E1 -9105.286,E2 -9105.286} C_VEL
LIN {X 0,Y 440.526,Z 453.316,A -85,B 0,C 180,E1 -9105.874,E2 -9105.874} C_VEL
LIN {X 0,Y 439.23,Z 440.23,A -85,B 0,C 180,E1 -9106.299,E2 -9106.299} C_VEL
LIN {X 0,Y 438.944,Z 437.176,A -85,B 0,C 180,E1 -9106.433,E2 -9106.433} C_VEL
LIN {X 0,Y 439.309,Z 423.986,A -85,B 0,C 180,E1 -9109.63,E2 -9109.63} C_VEL
LIN {X 0,Y 439.784,Z 410.197,A -85,B 0,C 180,E1 -9113.049,E2 -9113.049} C_VEL
LIN {X 0,Y 440.281,Z 398.322,A -85,B 0,C 180,E1 -9116.037,E2 -9116.037} C_VEL
LIN {X 0,Y 440.801,Z 386.373,A -85,B 0,C 180,E1 -9119.114,E2 -9119.114} C_VEL
LIN {X 0,Y 441.465,Z 375.038,A -85,B 0,C 180,E1 -9122.088,E2 -9122.088} C_VEL
LIN {X 0,Y 442.598,Z 360.613,A -85,B 0,C 180,E1 -9125.98,E2 -9125.98} C_VEL
LIN {X 0,Y 442.515,Z 356.57,A -85,B 0,C 180,E1 -9127.121,E2 -9127.121} C_VEL
LIN {X 0,Y 440.615,Z 346.945,A -85,B 0,C 180,E1 -9130.038,E2 -9130.038} C_VEL
LIN {X 0,Y 439.375,Z 340.838,A -85,B 0,C 180,E1 -9132.015,E2 -9132.015} C_VEL
LIN {X 0,Y 439.392,Z 340.756,A -85,B 0,C 180,E1 -9135.269,E2 -9135.269} C_VEL
LIN {X 0,Y 439.349,Z 340.757,A -85,B 0,C 180,E1 -9139.016,E2 -9139.016} C_VEL
LIN {X 0,Y 439.339,Z 340.755,A -85,B 0,C 180,E1 -9142.564,E2 -9142.564} C_VEL
LIN {X 0,Y 439.389,Z 340.751,A -85,B 0,C 180,E1 -9144.843,E2 -9144.843} C_VEL
LIN {X 0,Y 439.363,Z 340.752,A -85,B 0,C 180,E1 -9148.139,E2 -9148.139} C_VEL
LIN {X 0,Y 439.425,Z 340.747,A -85,B 0,C 180,E1 -9151.597,E2 -9151.597} C_VEL
LIN {X 0,Y 439.388,Z 340.749,A -85,B 0,C 180,E1 -9154.414,E2 -9154.414} C_VEL
LIN {X 0,Y 439.354,Z 340.757,A -85,B 0,C 180,E1 -9157.424,E2 -9157.424} C_VEL
LIN {X 0,Y 439.431,Z 340.746,A -85,B 0,C 180,E1 -9160.663,E2 -9160.663} C_VEL
LIN {X 0,Y 439.452,Z 340.741,A -85,B 0,C 180,E1 -9164.224,E2 -9164.224} C_VEL
LIN {X 0,Y 439.473,Z 340.738,A -85,B 0,C 180,E1 -9168.001,E2 -9168.001} C_VEL
LIN {X 0,Y 439.493,Z 340.736,A -85,B 0,C 180,E1 -9171.725,E2 -9171.725} C_VEL
LIN {X 0,Y 439.603,Z 340.725,A -85,B 0,C 180,E1 -9174.496,E2 -9174.496} C_VEL
LIN {X 0,Y 439.624,Z 340.72,A -85,B 0,C 180,E1 -9178.168,E2 -9178.168} C_VEL
LIN {X 0,Y 439.751,Z 340.704,A -85,B 0,C 180,E1 -9180,E2 -9180} C_VEL
LIN {X 0,Y 439.628,Z 340.726,A -85,B 0,C 180,E1 -9182.749,E2 -9182.749} C_VEL
LIN {X 0,Y 439.602,Z 340.726,A -85,B 0,C 180,E1 -9186.425,E2 -9186.425} C_VEL
LIN {X 0,Y 439.49,Z 340.738,A -85,B 0,C 180,E1 -9189.202,E2 -9189.202} C_VEL
LIN {X 0,Y 439.456,Z 340.744,A -85,B 0,C 180,E1 -9192.938,E2 -9192.938} C_VEL
LIN {X 0,Y 439.438,Z 340.747,A -85,B 0,C 180,E1 -9196.349,E2 -9196.349} C_VEL
LIN {X 0,Y 439.395,Z 340.748,A -85,B 0,C 180,E1 -9199.627,E2 -9199.627} C_VEL
LIN {X 0,Y 439.359,Z 340.759,A -85,B 0,C 180,E1 -9202.576,E2 -9202.576} C_VEL
LIN {X 0,Y 439.397,Z 340.748,A -85,B 0,C 180,E1 -9205.585,E2 -9205.585} C_VEL
LIN {X 0,Y 439.417,Z 340.749,A -85,B 0,C 180,E1 -9208.674,E2 -9208.674} C_VEL
LIN {X 0,Y 439.366,Z 340.753,A -85,B 0,C 180,E1 -9211.861,E2 -9211.861} C_VEL
LIN {X 0,Y 439.394,Z 340.748,A -85,B 0,C 180,E1 -9215.157,E2 -9215.157} C_VEL
LIN {X 0,Y 439.389,Z 340.752,A -85,B 0,C 180,E1 -9218.594,E2 -9218.594} C_VEL
LIN {X 0,Y 439.393,Z 340.748,A -85,B 0,C 180,E1 -9221.259,E2 -9221.259} C_VEL
LIN {X 0,Y 439.397,Z 340.749,A -85,B 0,C 180,E1 -9224.73,E2 -9224.73} C_VEL
LIN {X 0,Y 439.394,Z 340.751,A -85,B 0,C 180,E1 -9227.797,E2 -9227.797} C_VEL
LIN {X 0,Y 439.433,Z 340.749,A -85,B 0,C 180,E1 -9230.229,E2 -9230.229} C_VEL
LIN {X 0,Y 439.374,Z 340.754,A -85,B 0,C 180,E1 -9233.714,E2 -9233.714} C_VEL
LIN {X 0,Y 439.373,Z 340.75,A -85,B 0,C 180,E1 -9237.055,E2 -9237.055} C_VEL
LIN {X 0,Y 439.396,Z 340.751,A -85,B 0,C 180,E1 -9240.276,E2 -9240.276} C_VEL
LIN {X 0,Y 439.433,Z 340.747,A -85,B 0,C 180,E1 -9243.589,E2 -9243.589} C_VEL
LIN {X 0,Y 439.388,Z 340.75,A -85,B 0,C 180,E1 -9246.43,E2 -9246.43} C_VEL
LIN {X 0,Y 439.39,Z 340.751,A -85,B 0,C 180,E1 -9249.398,E2 -9249.398} C_VEL
LIN {X 0,Y 439.434,Z 340.745,A -85,B 0,C 180,E1 -9252.31,E2 -9252.31} C_VEL
LIN {X 0,Y 439.454,Z 340.742,A -85,B 0,C 180,E1 -9255.175,E2 -9255.175} C_VEL
LIN {X 0,Y 439.486,Z 340.74,A -85,B 0,C 180,E1 -9258.002,E2 -9258.002} C_VEL
LIN {X 0,Y 439.55,Z 340.735,A -85,B 0,C 180,E1 -9261.727,E2 -9261.727} C_VEL
LIN {X 0,Y 439.626,Z 340.719,A -85,B 0,C 180,E1 -9264.496,E2 -9264.496} C_VEL
LIN {X 0,Y 439.638,Z 340.719,A -85,B 0,C 180,E1 -9268.168,E2 -9268.168} C_VEL
LIN {X 0,Y 439.767,Z 340.704,A -85,B 0,C 180,E1 -9270,E2 -9270} C_VEL
LIN {X 0,Y 439.624,Z 340.72,A -85,B 0,C 180,E1 -9271.008,E2 -9271.008} C_VEL
LIN {X 0,Y 438.91,Z 340.813,A -85,B 0,C 180,E1 -9271.772,E2 -9271.772} C_VEL
LIN {X 0,Y 435.932,Z 341.181,A -85,B 0,C 180,E1 -9273.011,E2 -9273.011} C_VEL
LIN {X 0,Y 433.48,Z 341.486,A -85,B 0,C 180,E1 -9274.011,E2 -9274.011} C_VEL
LIN {X 0,Y 432.506,Z 341.607,A -85,B 0,C 180,E1 -9274.786,E2 -9274.786} C_VEL
LIN {X 0,Y 432.469,Z 341.611,A -85,B 0,C 180,E1 -9275.048,E2 -9275.048} C_VEL
LIN {X 0,Y 432.562,Z 341.604,A -85,B 0,C 180,E1 -9277.653,E2 -9277.653} C_VEL
LIN {X 0,Y 432.395,Z 341.626,A -85,B 0,C 180,E1 -9281.247,E2 -9281.247} C_VEL
LIN {X 0,Y 432.377,Z 341.622,A -85,B 0,C 180,E1 -9284.111,E2 -9284.111} C_VEL
LIN {X 0,Y 432.399,Z 341.623,A -85,B 0,C 180,E1 -9287.011,E2 -9287.011} C_VEL
LIN {X 0,Y 432.34,Z 341.627,A -85,B 0,C 180,E1 -9289.96,E2 -9289.96} C_VEL
LIN {X 0,Y 432.32,Z 341.633,A -85,B 0,C 180,E1 -9292.964,E2 -9292.964} C_VEL
LIN {X 0,Y 432.365,Z 341.624,A -85,B 0,C 180,E1 -9296.032,E2 -9296.032} C_VEL
LIN {X 0,Y 432.342,Z 341.633,A -85,B 0,C 180,E1 -9299.187,E2 -9299.187} C_VEL
LIN {X 0,Y 432.322,Z 341.63,A -85,B 0,C 180,E1 -9302.442,E2 -9302.442} C_VEL
LIN {X 0,Y 432.344,Z 341.627,A -85,B 0,C 180,E1 -9305.631,E2 -9305.631} C_VEL
LIN {X 0,Y 432.358,Z 341.628,A -85,B 0,C 180,E1 -9308.717,E2 -9308.717} C_VEL
LIN {X 0,Y 432.37,Z 341.626,A -85,B 0,C 180,E1 -9311.791,E2 -9311.791} C_VEL
LIN {X 0,Y 432.374,Z 341.628,A -85,B 0,C 180,E1 -9314.341,E2 -9314.341} C_VEL
LIN {X 0,Y 432.401,Z 341.771,A -85,B 0,C 180,E1 -9316.324,E2 -9316.324} C_VEL
LIN {X 0,Y 432.672,Z 342.926,A -85,B 0,C 180,E1 -9316.497,E2 -9316.497} C_VEL
LIN {X 0,Y 435.617,Z 353.191,A -85,B 0,C 180,E1 -9317.23,E2 -9317.23} C_VEL
LIN {X 0,Y 435.69,Z 359.641,A -85,B 0,C 180,E1 -9317.699,E2 -9317.699} C_VEL
LIN {X 0,Y 435.127,Z 371.049,A -85,B 0,C 180,E1 -9318.663,E2 -9318.663} C_VEL
LIN {X 0,Y 434.607,Z 380.898,A -85,B 0,C 180,E1 -9319.696,E2 -9319.696} C_VEL
LIN {X 0,Y 434.013,Z 390.95,A -85,B 0,C 180,E1 -9321.009,E2 -9321.009} C_VEL
LIN {X 0,Y 433.538,Z 399.246,A -85,B 0,C 180,E1 -9322.346,E2 -9322.346} C_VEL
LIN {X 0,Y 433.147,Z 405.977,A -85,B 0,C 180,E1 -9323.685,E2 -9323.685} C_VEL
LIN {X 0,Y 432.708,Z 412.58,A -85,B 0,C 180,E1 -9325.357,E2 -9325.357} C_VEL
LIN {X 0,Y 432.469,Z 417.527,A -85,B 0,C 180,E1 -9327.016,E2 -9327.016} C_VEL
LIN {X 0,Y 432.304,Z 420.935,A -85,B 0,C 180,E1 -9328.652,E2 -9328.652} C_VEL
LIN {X 0,Y 432.209,Z 422.494,A -85,B 0,C 180,E1 -9329.73,E2 -9329.73} C_VEL
LIN {X 0,Y 432.129,Z 423.861,A -85,B 0,C 180,E1 -9331.428,E2 -9331.428} C_VEL
LIN {X 0,Y 432.169,Z 423.768,A -85,B 0,C 180,E1 -9333.431,E2 -9333.431} C_VEL
LIN {X 0,Y 432.356,Z 422.427,A -85,B 0,C 180,E1 -9334.999,E2 -9334.999} C_VEL
LIN {X 0,Y 432.579,Z 419.967,A -85,B 0,C 180,E1 -9336.544,E2 -9336.544} C_VEL
LIN {X 0,Y 432.886,Z 416.339,A -85,B 0,C 180,E1 -9338.074,E2 -9338.074} C_VEL
LIN {X 0,Y 433.274,Z 411.478,A -85,B 0,C 180,E1 -9339.589,E2 -9339.589} C_VEL
LIN {X 0,Y 433.69,Z 405.283,A -85,B 0,C 180,E1 -9341.089,E2 -9341.089} C_VEL
LIN {X 0,Y 434.255,Z 398.107,A -85,B 0,C 180,E1 -9342.459,E2 -9342.459} C_VEL
LIN {X 0,Y 434.847,Z 389.297,A -85,B 0,C 180,E1 -9343.812,E2 -9343.812} C_VEL
LIN {X 0,Y 435.516,Z 379.382,A -85,B 0,C 180,E1 -9345.037,E2 -9345.037} C_VEL
LIN {X 0,Y 436.156,Z 368.171,A -85,B 0,C 180,E1 -9346.132,E2 -9346.132} C_VEL
LIN {X 0,Y 436.677,Z 357.289,A -85,B 0,C 180,E1 -9346.978,E2 -9346.978} C_VEL
LIN {X 0,Y 436.294,Z 354.249,A -85,B 0,C 180,E1 -9347.203,E2 -9347.203} C_VEL
LIN {X 0,Y 432.597,Z 342.346,A -85,B 0,C 180,E1 -9348.105,E2 -9348.105} C_VEL
LIN {X 0,Y 432.439,Z 341.643,A -85,B 0,C 180,E1 -9348.338,E2 -9348.338} C_VEL
LIN {X 0,Y 432.553,Z 341.604,A -85,B 0,C 180,E1 -9352.344,E2 -9352.344} C_VEL
LIN {X 0,Y 432.582,Z 341.6,A -85,B 0,C 180,E1 -9354.406,E2 -9354.406} C_VEL
LIN {X 0,Y 432.592,Z 341.598,A -85,B 0,C 180,E1 -9358.138,E2 -9358.138} C_VEL
LIN {X 0,Y 432.722,Z 341.583,A -85,B 0,C 180,E1 -9360,E2 -9360} C_VEL
LIN {X 0,Y 432.58,Z 341.601,A -85,B 0,C 180,E1 -9362.794,E2 -9362.794} C_VEL
LIN {X 0,Y 432.544,Z 341.604,A -85,B 0,C 180,E1 -9366.531,E2 -9366.531} C_VEL
LIN {X 0,Y 432.429,Z 341.621,A -85,B 0,C 180,E1 -9369.353,E2 -9369.353} C_VEL
LIN {X 0,Y 432.421,Z 341.621,A -85,B 0,C 180,E1 -9372.804,E2 -9372.804} C_VEL
LIN {X 0,Y 432.402,Z 341.622,A -85,B 0,C 180,E1 -9376.479,E2 -9376.479} C_VEL
LIN {X 0,Y 432.329,Z 341.629,A -85,B 0,C 180,E1 -9379.961,E2 -9379.961} C_VEL
LIN {X 0,Y 432.309,Z 341.635,A -85,B 0,C 180,E1 -9382.965,E2 -9382.965} C_VEL
LIN {X 0,Y 432.353,Z 341.625,A -85,B 0,C 180,E1 -9386.033,E2 -9386.033} C_VEL
LIN {X 0,Y 432.334,Z 341.632,A -85,B 0,C 180,E1 -9389.188,E2 -9389.188} C_VEL
LIN {X 0,Y 432.315,Z 341.635,A -85,B 0,C 180,E1 -9392.444,E2 -9392.444} C_VEL
LIN {X 0,Y 432.336,Z 341.63,A -85,B 0,C 180,E1 -9395.632,E2 -9395.632} C_VEL
LIN {X 0,Y 432.319,Z 341.635,A -85,B 0,C 180,E1 -9398.713,E2 -9398.713} C_VEL
LIN {X 0,Y 432.299,Z 341.635,A -85,B 0,C 180,E1 -9401.801,E2 -9401.801} C_VEL
LIN {X 0,Y 432.328,Z 341.63,A -85,B 0,C 180,E1 -9404.348,E2 -9404.348} C_VEL
LIN {X 0,Y 432.302,Z 341.638,A -85,B 0,C 180,E1 -9407.019,E2 -9407.019} C_VEL
LIN {X 0,Y 432.356,Z 341.806,A -85,B 0,C 180,E1 -9408.395,E2 -9408.395} C_VEL
LIN {X 0,Y 434.17,Z 350.785,A -85,B 0,C 180,E1 -9411.557,E2 -9411.557} C_VEL
LIN {X 0,Y 435.041,Z 356.161,A -85,B 0,C 180,E1 -9413.294,E2 -9413.294} C_VEL
LIN {X 0,Y 434.796,Z 359.958,A -85,B 0,C 180,E1 -9414.417,E2 -9414.417} C_VEL
LIN {X 0,Y 433.806,Z 373.524,A -85,B 0,C 180,E1 -9418.23,E2 -9418.23} C_VEL
LIN {X 0,Y 433.232,Z 385.904,A -85,B 0,C 180,E1 -9421.539,E2 -9421.539} C_VEL
LIN {X 0,Y 432.67,Z 399.463,A -85,B 0,C 180,E1 -9425.019,E2 -9425.019} C_VEL
LIN {X 0,Y 432.264,Z 413.612,A -85,B 0,C 180,E1 -9428.543,E2 -9428.543} C_VEL
LIN {X 0,Y 431.997,Z 427.8,A -85,B 0,C 180,E1 -9431.995,E2 -9431.995} C_VEL
LIN {X 0,Y 431.895,Z 432.623,A -85,B 0,C 180,E1 -9433.101,E2 -9433.101} C_VEL
LIN {X 0,Y 432.306,Z 436.508,A -85,B 0,C 180,E1 -9433.262,E2 -9433.262} C_VEL
LIN {X 0,Y 433.569,Z 449.847,A -85,B 0,C 180,E1 -9433.732,E2 -9433.732} C_VEL
LIN {X 0,Y 434.216,Z 462.466,A -85,B 0,C 180,E1 -9434.33,E2 -9434.33} C_VEL
LIN {X 0,Y 434.622,Z 469.796,A -85,B 0,C 180,E1 -9434.766,E2 -9434.766} C_VEL
LIN {X 0,Y 433.919,Z 481.698,A -85,B 0,C 180,E1 -9435.581,E2 -9435.581} C_VEL
LIN {X 0,Y 433.242,Z 493.016,A -85,B 0,C 180,E1 -9436.562,E2 -9436.562} C_VEL
LIN {X 0,Y 432.867,Z 502.657,A -85,B 0,C 180,E1 -9437.59,E2 -9437.59} C_VEL
LIN {X 0,Y 432.299,Z 511.707,A -85,B 0,C 180,E1 -9438.75,E2 -9438.75} C_VEL
LIN {X 0,Y 431.864,Z 520.741,A -85,B 0,C 180,E1 -9440.162,E2 -9440.162} C_VEL
LIN {X 0,Y 431.697,Z 528.019,A -85,B 0,C 180,E1 -9441.575,E2 -9441.575} C_VEL
LIN {X 0,Y 431.644,Z 534.069,A -85,B 0,C 180,E1 -9443.033,E2 -9443.033} C_VEL
LIN {X 0,Y 431.667,Z 538.542,A -85,B 0,C 180,E1 -9444.394,E2 -9444.394} C_VEL
LIN {X 0,Y 431.784,Z 542.078,A -85,B 0,C 180,E1 -9445.8,E2 -9445.8} C_VEL
LIN {X 0,Y 431.767,Z 544.563,A -85,B 0,C 180,E1 -9447.201,E2 -9447.201} C_VEL
LIN {X 0,Y 431.97,Z 546.395,A -85,B 0,C 180,E1 -9449.068,E2 -9449.068} C_VEL
LIN {X 0,Y 431.969,Z 546.661,A -85,B 0,C 180,E1 -9450,E2 -9450} C_VEL
LIN {X 0,Y 431.965,Z 546.482,A -85,B 0,C 180,E1 -9450.932,E2 -9450.932} C_VEL
LIN {X 0,Y 431.737,Z 544.876,A -85,B 0,C 180,E1 -9452.799,E2 -9452.799} C_VEL
LIN {X 0,Y 431.754,Z 543.425,A -85,B 0,C 180,E1 -9453.733,E2 -9453.733} C_VEL
LIN {X 0,Y 431.683,Z 540.396,A -85,B 0,C 180,E1 -9455.137,E2 -9455.137} C_VEL
LIN {X 0,Y 431.664,Z 535.707,A -85,B 0,C 180,E1 -9456.707,E2 -9456.707} C_VEL
LIN {X 0,Y 431.688,Z 528.899,A -85,B 0,C 180,E1 -9458.425,E2 -9458.425} C_VEL
LIN {X 0,Y 431.84,Z 521.682,A -85,B 0,C 180,E1 -9459.839,E2 -9459.839} C_VEL
LIN {X 0,Y 432.299,Z 512.754,A -85,B 0,C 180,E1 -9461.25,E2 -9461.25} C_VEL
LIN {X 0,Y 432.886,Z 503.733,A -85,B 0,C 180,E1 -9462.41,E2 -9462.41} C_VEL
LIN {X 0,Y 433.31,Z 493.896,A -85,B 0,C 180,E1 -9463.446,E2 -9463.446} C_VEL
LIN {X 0,Y 433.948,Z 482.432,A -85,B 0,C 180,E1 -9464.418,E2 -9464.418} C_VEL
LIN {X 0,Y 434.648,Z 470.171,A -85,B 0,C 180,E1 -9465.233,E2 -9465.233} C_VEL
LIN {X 0,Y 433.86,Z 456.853,A -85,B 0,C 180,E1 -9465.924,E2 -9465.924} C_VEL
LIN {X 0,Y 432.619,Z 443.486,A -85,B 0,C 180,E1 -9466.434,E2 -9466.434} C_VEL
LIN {X 0,Y 431.878,Z 436.525,A -85,B 0,C 180,E1 -9466.663,E2 -9466.663} C_VEL
LIN {X 0,Y 432.188,Z 426.984,A -85,B 0,C 180,E1 -9468.979,E2 -9468.979} C_VEL
LIN {X 0,Y 432.688,Z 411.259,A -85,B 0,C 180,E1 -9472.943,E2 -9472.943} C_VEL
LIN {X 0,Y 433.305,Z 397.703,A -85,B 0,C 180,E1 -9476.429,E2 -9476.429} C_VEL
LIN {X 0,Y 434.044,Z 383.624,A -85,B 0,C 180,E1 -9480.128,E2 -9480.128} C_VEL
LIN {X 0,Y 434.913,Z 369.738,A -85,B 0,C 180,E1 -9483.882,E2 -9483.882} C_VEL
LIN {X 0,Y 435.746,Z 359.81,A -85,B 0,C 180,E1 -9486.637,E2 -9486.637} C_VEL
LIN {X 0,Y 434.716,Z 353.759,A -85,B 0,C 180,E1 -9488.456,E2 -9488.456} C_VEL
LIN {X 0,Y 432.703,Z 343.633,A -85,B 0,C 180,E1 -9491.657,E2 -9491.657} C_VEL
LIN {X 0,Y 432.309,Z 341.7,A -85,B 0,C 180,E1 -9492.357,E2 -9492.357} C_VEL
LIN {X 0,Y 432.328,Z 341.635,A -85,B 0,C 180,E1 -9495.664,E2 -9495.664} C_VEL
LIN {X 0,Y 432.305,Z 341.632,A -85,B 0,C 180,E1 -9498.401,E2 -9498.401} C_VEL
LIN {X 0,Y 432.323,Z 341.63,A -85,B 0,C 180,E1 -9501.848,E2 -9501.848} C_VEL
LIN {X 0,Y 432.33,Z 341.635,A -85,B 0,C 180,E1 -9505.322,E2 -9505.322} C_VEL
LIN {X 0,Y 432.312,Z 341.631,A -85,B 0,C 180,E1 -9508.653,E2 -9508.653} C_VEL
LIN {X 0,Y 432.373,Z 341.623,A -85,B 0,C 180,E1 -9511.876,E2 -9511.876} C_VEL
LIN {X 0,Y 432.337,Z 341.633,A -85,B 0,C 180,E1 -9514.998,E2 -9514.998} C_VEL
LIN {X 0,Y 432.348,Z 341.626,A -85,B 0,C 180,E1 -9518.045,E2 -9518.045} C_VEL
LIN {X 0,Y 432.375,Z 341.629,A -85,B 0,C 180,E1 -9521.029,E2 -9521.029} C_VEL
LIN {X 0,Y 432.42,Z 341.617,A -85,B 0,C 180,E1 -9523.961,E2 -9523.961} C_VEL
LIN {X 0,Y 432.449,Z 341.613,A -85,B 0,C 180,E1 -9527.803,E2 -9527.803} C_VEL
LIN {X 0,Y 432.454,Z 341.613,A -85,B 0,C 180,E1 -9531.59,E2 -9531.59} C_VEL
LIN {X 0,Y 432.58,Z 341.599,A -85,B 0,C 180,E1 -9534.406,E2 -9534.406} C_VEL
LIN {X 0,Y 432.594,Z 341.596,A -85,B 0,C 180,E1 -9538.138,E2 -9538.138} C_VEL
LIN {X 0,Y 432.722,Z 341.579,A -85,B 0,C 180,E1 -9540,E2 -9540} C_VEL
LIN {X 0,Y 432.58,Z 341.604,A -85,B 0,C 180,E1 -9542.794,E2 -9542.794} C_VEL
LIN {X 0,Y 432.558,Z 341.605,A -85,B 0,C 180,E1 -9546.531,E2 -9546.531} C_VEL
LIN {X 0,Y 432.433,Z 341.616,A -85,B 0,C 180,E1 -9549.353,E2 -9549.353} C_VEL
LIN {X 0,Y 432.421,Z 341.622,A -85,B 0,C 180,E1 -9552.804,E2 -9552.804} C_VEL
LIN {X 0,Y 432.403,Z 341.625,A -85,B 0,C 180,E1 -9556.479,E2 -9556.479} C_VEL
LIN {X 0,Y 432.332,Z 341.629,A -85,B 0,C 180,E1 -9559.961,E2 -9559.961} C_VEL
LIN {X 0,Y 432.312,Z 341.632,A -85,B 0,C 180,E1 -9562.965,E2 -9562.965} C_VEL
LIN {X 0,Y 432.356,Z 341.627,A -85,B 0,C 180,E1 -9566.033,E2 -9566.033} C_VEL
LIN {X 0,Y 432.345,Z 341.626,A -85,B 0,C 180,E1 -9569.187,E2 -9569.187} C_VEL
LIN {X 0,Y 432.318,Z 341.636,A -85,B 0,C 180,E1 -9572.294,E2 -9572.294} C_VEL
LIN {X 0,Y 432.334,Z 341.631,A -85,B 0,C 180,E1 -9574.678,E2 -9574.678} C_VEL
LIN {X 0,Y 432.344,Z 341.632,A -85,B 0,C 180,E1 -9578.149,E2 -9578.149} C_VEL
LIN {X 0,Y 432.361,Z 341.625,A -85,B 0,C 180,E1 -9581.608,E2 -9581.608} C_VEL
LIN {X 0,Y 432.329,Z 341.633,A -85,B 0,C 180,E1 -9584.348,E2 -9584.348} C_VEL
LIN {X 0,Y 432.321,Z 341.629,A -85,B 0,C 180,E1 -9587.016,E2 -9587.016} C_VEL
LIN {X 0,Y 432.338,Z 341.631,A -85,B 0,C 180,E1 -9589.82,E2 -9589.82} C_VEL
LIN {X 0,Y 432.313,Z 341.63,A -85,B 0,C 180,E1 -9593.024,E2 -9593.024} C_VEL
LIN {X 0,Y 432.358,Z 341.632,A -85,B 0,C 180,E1 -9595.997,E2 -9595.997} C_VEL
LIN {X 0,Y 432.394,Z 341.625,A -85,B 0,C 180,E1 -9599.745,E2 -9599.745} C_VEL
LIN {X 0,Y 432.4,Z 341.621,A -85,B 0,C 180,E1 -9603.373,E2 -9603.373} C_VEL
LIN {X 0,Y 432.372,Z 341.628,A -85,B 0,C 180,E1 -9606.024,E2 -9606.024} C_VEL
LIN {X 0,Y 432.351,Z 341.625,A -85,B 0,C 180,E1 -9609.047,E2 -9609.047} C_VEL
LIN {X 0,Y 432.38,Z 341.626,A -85,B 0,C 180,E1 -9612.012,E2 -9612.012} C_VEL
LIN {X 0,Y 432.404,Z 341.619,A -85,B 0,C 180,E1 -9614.927,E2 -9614.927} C_VEL
LIN {X 0,Y 432.461,Z 341.618,A -85,B 0,C 180,E1 -9617.804,E2 -9617.804} C_VEL
LIN {X 0,Y 432.494,Z 341.614,A -85,B 0,C 180,E1 -9621.591,E2 -9621.591} C_VEL
LIN {X 0,Y 432.602,Z 341.594,A -85,B 0,C 180,E1 -9624.406,E2 -9624.406} C_VEL
LIN {X 0,Y 432.608,Z 341.595,A -85,B 0,C 180,E1 -9628.138,E2 -9628.138} C_VEL
LIN {X 0,Y 432.737,Z 341.579,A -85,B 0,C 180,E1 -9630,E2 -9630} C_VEL
LIN {X 0,Y 432.608,Z 341.594,A -85,B 0,C 180,E1 -9632.793,E2 -9632.793} C_VEL
LIN {X 0,Y 432.469,Z 341.611,A -85,B 0,C 180,E1 -9635.048,E2 -9635.048} C_VEL
LIN {X 0,Y 431.909,Z 341.686,A -85,B 0,C 180,E1 -9635.826,E2 -9635.826} C_VEL
LIN {X 0,Y 429.061,Z 342.038,A -85,B 0,C 180,E1 -9637.09,E2 -9637.09} C_VEL
LIN {X 0,Y 426.576,Z 342.345,A -85,B 0,C 180,E1 -9638.111,E2 -9638.111} C_VEL
LIN {X 0,Y 425.495,Z 342.481,A -85,B 0,C 180,E1 -9638.9,E2 -9638.9} C_VEL
LIN {X 0,Y 425.404,Z 342.493,A -85,B 0,C 180,E1 -9639.168,E2 -9639.168} C_VEL
LIN {X 0,Y 425.395,Z 342.494,A -85,B 0,C 180,E1 -9642.903,E2 -9642.903} C_VEL
LIN {X 0,Y 425.363,Z 342.496,A -85,B 0,C 180,E1 -9646.605,E2 -9646.605} C_VEL
LIN {X 0,Y 425.33,Z 342.503,A -85,B 0,C 180,E1 -9649.635,E2 -9649.635} C_VEL
LIN {X 0,Y 425.308,Z 342.508,A -85,B 0,C 180,E1 -9653.364,E2 -9653.364} C_VEL
LIN {X 0,Y 425.348,Z 342.501,A -85,B 0,C 180,E1 -9656.844,E2 -9656.844} C_VEL
LIN {X 0,Y 425.29,Z 342.506,A -85,B 0,C 180,E1 -9659.719,E2 -9659.719} C_VEL
LIN {X 0,Y 425.281,Z 342.513,A -85,B 0,C 180,E1 -9663.047,E2 -9663.047} C_VEL
LIN {X 0,Y 425.283,Z 342.506,A -85,B 0,C 180,E1 -9665.929,E2 -9665.929} C_VEL
LIN {X 0,Y 425.311,Z 342.509,A -85,B 0,C 180,E1 -9669.045,E2 -9669.045} C_VEL
LIN {X 0,Y 425.328,Z 342.505,A -85,B 0,C 180,E1 -9672.645,E2 -9672.645} C_VEL
LIN {X 0,Y 425.401,Z 342.734,A -85,B 0,C 180,E1 -9676.117,E2 -9676.117} C_VEL
LIN {X 0,Y 425.623,Z 343.83,A -85,B 0,C 180,E1 -9676.266,E2 -9676.266} C_VEL
LIN {X 0,Y 428.618,Z 354.348,A -85,B 0,C 180,E1 -9677.028,E2 -9677.028} C_VEL
LIN {X 0,Y 428.938,Z 356.974,A -85,B 0,C 180,E1 -9677.229,E2 -9677.229} C_VEL
LIN {X 0,Y 428.495,Z 367.459,A -85,B 0,C 180,E1 -9678.059,E2 -9678.059} C_VEL
LIN {X 0,Y 427.965,Z 377.708,A -85,B 0,C 180,E1 -9679.059,E2 -9679.059} C_VEL
LIN {X 0,Y 427.369,Z 387.719,A -85,B 0,C 180,E1 -9680.271,E2 -9680.271} C_VEL
LIN {X 0,Y 426.809,Z 396.324,A -85,B 0,C 180,E1 -9681.547,E2 -9681.547} C_VEL
LIN {X 0,Y 426.288,Z 404.276,A -85,B 0,C 180,E1 -9683.004,E2 -9683.004} C_VEL
LIN {X 0,Y 425.979,Z 410.054,A -85,B 0,C 180,E1 -9684.32,E2 -9684.32} C_VEL
LIN {X 0,Y 425.583,Z 415.392,A -85,B 0,C 180,E1 -9685.842,E2 -9685.842} C_VEL
LIN {X 0,Y 425.425,Z 419.535,A -85,B 0,C 180,E1 -9687.405,E2 -9687.405} C_VEL
LIN {X 0,Y 425.214,Z 422.908,A -85,B 0,C 180,E1 -9689.254,E2 -9689.254} C_VEL
LIN {X 0,Y 425.119,Z 424.74,A -85,B 0,C 180,E1 -9691.183,E2 -9691.183} C_VEL
LIN {X 0,Y 425.129,Z 425.042,A -85,B 0,C 180,E1 -9692.427,E2 -9692.427} C_VEL
LIN {X 0,Y 425.168,Z 424.785,A -85,B 0,C 180,E1 -9693.493,E2 -9693.493} C_VEL
LIN {X 0,Y 425.383,Z 423.123,A -85,B 0,C 180,E1 -9695.321,E2 -9695.321} C_VEL
LIN {X 0,Y 425.591,Z 420.98,A -85,B 0,C 180,E1 -9696.651,E2 -9696.651} C_VEL
LIN {X 0,Y 425.924,Z 417.356,A -85,B 0,C 180,E1 -9698.206,E2 -9698.206} C_VEL
LIN {X 0,Y 426.422,Z 411.761,A -85,B 0,C 180,E1 -9699.953,E2 -9699.953} C_VEL
LIN {X 0,Y 426.929,Z 405.094,A -85,B 0,C 180,E1 -9701.525,E2 -9701.525} C_VEL
LIN {X 0,Y 427.564,Z 396.929,A -85,B 0,C 180,E1 -9703.037,E2 -9703.037} C_VEL
LIN {X 0,Y 428.204,Z 388.504,A -85,B 0,C 180,E1 -9704.288,E2 -9704.288} C_VEL
LIN {X 0,Y 428.867,Z 378.856,A -85,B 0,C 180,E1 -9705.444,E2 -9705.444} C_VEL
LIN {X 0,Y 429.48,Z 367.805,A -85,B 0,C 180,E1 -9706.515,E2 -9706.515} C_VEL
LIN {X 0,Y 429.973,Z 358.274,A -85,B 0,C 180,E1 -9707.252,E2 -9707.252} C_VEL
LIN {X 0,Y 428.2,Z 351.393,A -85,B 0,C 180,E1 -9707.801,E2 -9707.801} C_VEL
LIN {X 0,Y 425.486,Z 343.111,A -85,B 0,C 180,E1 -9708.447,E2 -9708.447} C_VEL
LIN {X 0,Y 425.374,Z 342.516,A -85,B 0,C 180,E1 -9708.685,E2 -9708.685} C_VEL
LIN {X 0,Y 425.529,Z 342.48,A -85,B 0,C 180,E1 -9712.407,E2 -9712.407} C_VEL
LIN {X 0,Y 425.539,Z 342.478,A -85,B 0,C 180,E1 -9714.313,E2 -9714.313} C_VEL
LIN {X 0,Y 425.561,Z 342.474,A -85,B 0,C 180,E1 -9718.107,E2 -9718.107} C_VEL
LIN {X 0,Y 425.691,Z 342.459,A -85,B 0,C 180,E1 -9720,E2 -9720} C_VEL
LIN {X 0,Y 425.534,Z 342.479,A -85,B 0,C 180,E1 -9722.84,E2 -9722.84} C_VEL
LIN {X 0,Y 425.535,Z 342.479,A -85,B 0,C 180,E1 -9725.687,E2 -9725.687} C_VEL
LIN {X 0,Y 425.398,Z 342.493,A -85,B 0,C 180,E1 -9728.551,E2 -9728.551} C_VEL
LIN {X 0,Y 425.402,Z 342.492,A -85,B 0,C 180,E1 -9732.402,E2 -9732.402} C_VEL
LIN {X 0,Y 425.378,Z 342.496,A -85,B 0,C 180,E1 -9736.312,E2 -9736.312} C_VEL
LIN {X 0,Y 425.319,Z 342.503,A -85,B 0,C 180,E1 -9739.636,E2 -9739.636} C_VEL
LIN {X 0,Y 425.279,Z 342.509,A -85,B 0,C 180,E1 -9742.339,E2 -9742.339} C_VEL
LIN {X 0,Y 425.283,Z 342.508,A -85,B 0,C 180,E1 -9745.446,E2 -9745.446} C_VEL
LIN {X 0,Y 425.34,Z 342.502,A -85,B 0,C 180,E1 -9747.558,E2 -9747.558} C_VEL
LIN {X 0,Y 425.28,Z 342.511,A -85,B 0,C 180,E1 -9750.817,E2 -9750.817} C_VEL
LIN {X 0,Y 425.302,Z 342.507,A -85,B 0,C 180,E1 -9754.288,E2 -9754.288} C_VEL
LIN {X 0,Y 425.27,Z 342.512,A -85,B 0,C 180,E1 -9757.695,E2 -9757.695} C_VEL
LIN {X 0,Y 425.237,Z 342.517,A -85,B 0,C 180,E1 -9760.515,E2 -9760.515} C_VEL
LIN {X 0,Y 425.241,Z 342.517,A -85,B 0,C 180,E1 -9763.35,E2 -9763.35} C_VEL
LIN {X 0,Y 425.253,Z 342.513,A -85,B 0,C 180,E1 -9766.044,E2 -9766.044} C_VEL
LIN {X 0,Y 425.298,Z 342.675,A -85,B 0,C 180,E1 -9767.988,E2 -9767.988} C_VEL
LIN {X 0,Y 426.791,Z 350.085,A -85,B 0,C 180,E1 -9770.711,E2 -9770.711} C_VEL
LIN {X 0,Y 428.082,Z 357.288,A -85,B 0,C 180,E1 -9773.131,E2 -9773.131} C_VEL
LIN {X 0,Y 427.841,Z 361.251,A -85,B 0,C 180,E1 -9774.329,E2 -9774.329} C_VEL
LIN {X 0,Y 426.814,Z 374.746,A -85,B 0,C 180,E1 -9778.203,E2 -9778.203} C_VEL
LIN {X 0,Y 426.205,Z 386.582,A -85,B 0,C 180,E1 -9781.433,E2 -9781.433} C_VEL
LIN {X 0,Y 425.683,Z 398.555,A -85,B 0,C 180,E1 -9784.58,E2 -9784.58} C_VEL
LIN {X 0,Y 425.254,Z 410.942,A -85,B 0,C 180,E1 -9787.743,E2 -9787.743} C_VEL
LIN {X 0,Y 424.97,Z 423.717,A -85,B 0,C 180,E1 -9790.937,E2 -9790.937} C_VEL
LIN {X 0,Y 424.829,Z 431.339,A -85,B 0,C 180,E1 -9792.762,E2 -9792.762} C_VEL
LIN {X 0,Y 425.071,Z 433.729,A -85,B 0,C 180,E1 -9792.887,E2 -9792.887} C_VEL
LIN {X 0,Y 426.561,Z 447.919,A -85,B 0,C 180,E1 -9793.396,E2 -9793.396} C_VEL
LIN {X 0,Y 427.13,Z 460.653,A -85,B 0,C 180,E1 -9794.002,E2 -9794.002} C_VEL
LIN {X 0,Y 427.627,Z 470.897,A -85,B 0,C 180,E1 -9794.633,E2 -9794.633} C_VEL
LIN {X 0,Y 426.772,Z 483.689,A -85,B 0,C 180,E1 -9795.578,E2 -9795.578} C_VEL
LIN {X 0,Y 426.086,Z 495.169,A -85,B 0,C 180,E1 -9796.649,E2 -9796.649} C_VEL
LIN {X 0,Y 425.733,Z 503.579,A -85,B 0,C 180,E1 -9797.608,E2 -9797.608} C_VEL
LIN {X 0,Y 425.182,Z 512.399,A -85,B 0,C 180,E1 -9798.801,E2 -9798.801} C_VEL
LIN {X 0,Y 424.784,Z 521.047,A -85,B 0,C 180,E1 -9800.237,E2 -9800.237} C_VEL
LIN {X 0,Y 424.619,Z 528.086,A -85,B 0,C 180,E1 -9801.673,E2 -9801.673} C_VEL
LIN {X 0,Y 424.581,Z 534.593,A -85,B 0,C 180,E1 -9803.346,E2 -9803.346} C_VEL
LIN {X 0,Y 424.656,Z 538.856,A -85,B 0,C 180,E1 -9804.778,E2 -9804.778} C_VEL
LIN {X 0,Y 424.744,Z 542.037,A -85,B 0,C 180,E1 -9806.205,E2 -9806.205} C_VEL
LIN {X 0,Y 424.723,Z 543.558,A -85,B 0,C 180,E1 -9807.155,E2 -9807.155} C_VEL
LIN {X 0,Y 424.945,Z 545.397,A -85,B 0,C 180,E1 -9809.052,E2 -9809.052} C_VEL
LIN {X 0,Y 424.948,Z 545.656,A -85,B 0,C 180,E1 -9810,E2 -9810} C_VEL
LIN {X 0,Y 424.94,Z 545.474,A -85,B 0,C 180,E1 -9810.948,E2 -9810.948} C_VEL
LIN {X 0,Y 424.695,Z 543.861,A -85,B 0,C 180,E1 -9812.846,E2 -9812.846} C_VEL
LIN {X 0,Y 424.714,Z 542.399,A -85,B 0,C 180,E1 -9813.795,E2 -9813.795} C_VEL
LIN {X 0,Y 424.62,Z 539.354,A -85,B 0,C 180,E1 -9815.223,E2 -9815.223} C_VEL
LIN {X 0,Y 424.602,Z 534.978,A -85,B 0,C 180,E1 -9816.723,E2 -9816.723} C_VEL
LIN {X 0,Y 424.61,Z 528.85,A -85,B 0,C 180,E1 -9818.327,E2 -9818.327} C_VEL
LIN {X 0,Y 424.756,Z 521.912,A -85,B 0,C 180,E1 -9819.764,E2 -9819.764} C_VEL
LIN {X 0,Y 425.182,Z 513.249,A -85,B 0,C 180,E1 -9821.199,E2 -9821.199} C_VEL
LIN {X 0,Y 425.742,Z 504.413,A -85,B 0,C 180,E1 -9822.392,E2 -9822.392} C_VEL
LIN {X 0,Y 426.221,Z 494.738,A -85,B 0,C 180,E1 -9823.468,E2 -9823.468} C_VEL
LIN {X 0,Y 426.798,Z 484.222,A -85,B 0,C 180,E1 -9824.422,E2 -9824.422} C_VEL
LIN {X 0,Y 427.556,Z 472.654,A -85,B 0,C 180,E1 -9825.248,E2 -9825.248} C_VEL
LIN {X 0,Y 427.459,Z 466.558,A -85,B 0,C 180,E1 -9825.618,E2 -9825.618} C_VEL
LIN {X 0,Y 426.559,Z 452.901,A -85,B 0,C 180,E1 -9826.301,E2 -9826.301} C_VEL
LIN {X 0,Y 425.151,Z 439.036,A -85,B 0,C 180,E1 -9826.789,E2 -9826.789} C_VEL
LIN {X 0,Y 424.791,Z 435.483,A -85,B 0,C 180,E1 -9826.937,E2 -9826.937} C_VEL
LIN {X 0,Y 425.164,Z 423.761,A -85,B 0,C 180,E1 -9829.883,E2 -9829.883} C_VEL
LIN {X 0,Y 425.695,Z 410.359,A -85,B 0,C 180,E1 -9833.342,E2 -9833.342} C_VEL
LIN {X 0,Y 426.305,Z 397.255,A -85,B 0,C 180,E1 -9836.774,E2 -9836.774} C_VEL
LIN {X 0,Y 427.135,Z 382.765,A -85,B 0,C 180,E1 -9840.668,E2 -9840.668} C_VEL
LIN {X 0,Y 428.046,Z 369.265,A -85,B 0,C 180,E1 -9844.399,E2 -9844.399} C_VEL
LIN {X 0,Y 428.786,Z 361.571,A -85,B 0,C 180,E1 -9846.569,E2 -9846.569} C_VEL
LIN {X 0,Y 427.93,Z 356.008,A -85,B 0,C 180,E1 -9848.26,E2 -9848.26} C_VEL
LIN {X 0,Y 426.067,Z 346.543,A -85,B 0,C 180,E1 -9851.284,E2 -9851.284} C_VEL
LIN {X 0,Y 425.294,Z 342.581,A -85,B 0,C 180,E1 -9852.649,E2 -9852.649} C_VEL
LIN {X 0,Y 425.253,Z 342.514,A -85,B 0,C 180,E1 -9856.043,E2 -9856.043} C_VEL
LIN {X 0,Y 425.244,Z 342.511,A -85,B 0,C 180,E1 -9858.618,E2 -9858.618} C_VEL
LIN {X 0,Y 425.274,Z 342.511,A -85,B 0,C 180,E1 -9861.098,E2 -9861.098} C_VEL
LIN {X 0,Y 425.291,Z 342.506,A -85,B 0,C 180,E1 -9864.663,E2 -9864.663} C_VEL
LIN {X 0,Y 425.256,Z 342.509,A -85,B 0,C 180,E1 -9868.072,E2 -9868.072} C_VEL
LIN {X 0,Y 425.323,Z 342.506,A -85,B 0,C 180,E1 -9871.367,E2 -9871.367} C_VEL
LIN {X 0,Y 425.345,Z 342.501,A -85,B 0,C 180,E1 -9873.505,E2 -9873.505} C_VEL
LIN {X 0,Y 425.275,Z 342.509,A -85,B 0,C 180,E1 -9876.633,E2 -9876.633} C_VEL
LIN {X 0,Y 425.286,Z 342.507,A -85,B 0,C 180,E1 -9879.694,E2 -9879.694} C_VEL
LIN {X 0,Y 425.324,Z 342.504,A -85,B 0,C 180,E1 -9882.697,E2 -9882.697} C_VEL
LIN {X 0,Y 425.338,Z 342.5,A -85,B 0,C 180,E1 -9885.65,E2 -9885.65} C_VEL
LIN {X 0,Y 425.34,Z 342.501,A -85,B 0,C 180,E1 -9888.564,E2 -9888.564} C_VEL
LIN {X 0,Y 425.496,Z 342.48,A -85,B 0,C 180,E1 -9892.31,E2 -9892.31} C_VEL
LIN {X 0,Y 425.535,Z 342.476,A -85,B 0,C 180,E1 -9894.313,E2 -9894.313} C_VEL
LIN {X 0,Y 425.563,Z 342.471,A -85,B 0,C 180,E1 -9898.107,E2 -9898.107} C_VEL
LIN {X 0,Y 425.691,Z 342.455,A -85,B 0,C 180,E1 -9900,E2 -9900} C_VEL
LIN {X 0,Y 425.534,Z 342.481,A -85,B 0,C 180,E1 -9902.84,E2 -9902.84} C_VEL
LIN {X 0,Y 425.517,Z 342.483,A -85,B 0,C 180,E1 -9906.639,E2 -9906.639} C_VEL
LIN {X 0,Y 425.391,Z 342.492,A -85,B 0,C 180,E1 -9909.51,E2 -9909.51} C_VEL
LIN {X 0,Y 425.384,Z 342.497,A -85,B 0,C 180,E1 -9912.904,E2 -9912.904} C_VEL
LIN {X 0,Y 425.352,Z 342.504,A -85,B 0,C 180,E1 -9916.605,E2 -9916.605} C_VEL
LIN {X 0,Y 425.32,Z 342.501,A -85,B 0,C 180,E1 -9919.636,E2 -9919.636} C_VEL
LIN {X 0,Y 425.3,Z 342.504,A -85,B 0,C 180,E1 -9923.366,E2 -9923.366} C_VEL
LIN {X 0,Y 425.339,Z 342.501,A -85,B 0,C 180,E1 -9926.845,E2 -9926.845} C_VEL
LIN {X 0,Y 425.311,Z 342.503,A -85,B 0,C 180,E1 -9929.718,E2 -9929.718} C_VEL
LIN {X 0,Y 425.275,Z 342.507,A -85,B 0,C 180,E1 -9933.049,E2 -9933.049} C_VEL
LIN {X 0,Y 425.278,Z 342.509,A -85,B 0,C 180,E1 -9935.93,E2 -9935.93} C_VEL
LIN {X 0,Y 425.304,Z 342.503,A -85,B 0,C 180,E1 -9939.046,E2 -9939.046} C_VEL
LIN {X 0,Y 425.31,Z 342.507,A -85,B 0,C 180,E1 -9941.963,E2 -9941.963} C_VEL
LIN {X 0,Y 425.285,Z 342.506,A -85,B 0,C 180,E1 -9945.283,E2 -9945.283} C_VEL
LIN {X 0,Y 425.273,Z 342.509,A -85,B 0,C 180,E1 -9948.622,E2 -9948.622} C_VEL
LIN {X 0,Y 425.312,Z 342.502,A -85,B 0,C 180,E1 -9951.104,E2 -9951.104} C_VEL
LIN {X 0,Y 425.298,Z 342.505,A -85,B 0,C 180,E1 -9954.665,E2 -9954.665} C_VEL
LIN {X 0,Y 425.271,Z 342.514,A -85,B 0,C 180,E1 -9958.075,E2 -9958.075} C_VEL
LIN {X 0,Y 425.337,Z 342.5,A -85,B 0,C 180,E1 -9961.369,E2 -9961.369} C_VEL
LIN {X 0,Y 425.296,Z 342.505,A -85,B 0,C 180,E1 -9964.555,E2 -9964.555} C_VEL
LIN {X 0,Y 425.288,Z 342.51,A -85,B 0,C 180,E1 -9967.662,E2 -9967.662} C_VEL
LIN {X 0,Y 425.363,Z 342.496,A -85,B 0,C 180,E1 -9970.705,E2 -9970.705} C_VEL
LIN {X 0,Y 425.401,Z 342.498,A -85,B 0,C 180,E1 -9973.689,E2 -9973.689} C_VEL
LIN {X 0,Y 425.414,Z 342.495,A -85,B 0,C 180,E1 -9977.599,E2 -9977.599} C_VEL
LIN {X 0,Y 425.445,Z 342.49,A -85,B 0,C 180,E1 -9981.45,E2 -9981.45} C_VEL
LIN {X 0,Y 425.558,Z 342.472,A -85,B 0,C 180,E1 -9984.313,E2 -9984.313} C_VEL
LIN {X 0,Y 425.578,Z 342.471,A -85,B 0,C 180,E1 -9988.107,E2 -9988.107} C_VEL
LIN {X 0,Y 425.706,Z 342.455,A -85,B 0,C 180,E1 -9990,E2 -9990} C_VEL
LIN {X 0,Y 425.56,Z 342.472,A -85,B 0,C 180,E1 -9992.84,E2 -9992.84} C_VEL
LIN {X 0,Y 425.525,Z 342.476,A -85,B 0,C 180,E1 -9996.639,E2 -9996.639} C_VEL
LIN {X 0,Y 425.404,Z 342.493,A -85,B 0,C 180,E1 -9999.168,E2 -9999.168} C_VEL
LIN {X 0,Y 424.733,Z 342.581,A -85,B 0,C 180,E1 -9999.958,E2 -9999.958} C_VEL
LIN {X 0,Y 421.884,Z 342.936,A -85,B 0,C 180,E1 -10001.241,E2 -10001.241} C_VEL
LIN {X 0,Y 419.467,Z 343.234,A -85,B 0,C 180,E1 -10002.277,E2 -10002.277} C_VEL
LIN {X 0,Y 418.416,Z 343.365,A -85,B 0,C 180,E1 -10003.078,E2 -10003.078} C_VEL
LIN {X 0,Y 418.324,Z 343.376,A -85,B 0,C 180,E1 -10003.349,E2 -10003.349} C_VEL
LIN {X 0,Y 418.314,Z 343.375,A -85,B 0,C 180,E1 -10006.735,E2 -10006.735} C_VEL
LIN {X 0,Y 418.272,Z 343.381,A -85,B 0,C 180,E1 -10009.79,E2 -10009.79} C_VEL
LIN {X 0,Y 418.239,Z 343.385,A -85,B 0,C 180,E1 -10012.735,E2 -10012.735} C_VEL
LIN {X 0,Y 418.271,Z 343.38,A -85,B 0,C 180,E1 -10015.903,E2 -10015.903} C_VEL
LIN {X 0,Y 418.264,Z 343.387,A -85,B 0,C 180,E1 -10019.161,E2 -10019.161} C_VEL
LIN {X 0,Y 418.256,Z 343.385,A -85,B 0,C 180,E1 -10022.843,E2 -10022.843} C_VEL
LIN {X 0,Y 418.247,Z 343.382,A -85,B 0,C 180,E1 -10026.238,E2 -10026.238} C_VEL
LIN {X 0,Y 418.264,Z 343.384,A -85,B 0,C 180,E1 -10029.679,E2 -10029.679} C_VEL
LIN {X 0,Y 418.282,Z 343.382,A -85,B 0,C 180,E1 -10032.329,E2 -10032.329} C_VEL
LIN {X 0,Y 418.329,Z 343.588,A -85,B 0,C 180,E1 -10035.866,E2 -10035.866} C_VEL
LIN {X 0,Y 418.573,Z 344.667,A -85,B 0,C 180,E1 -10036.024,E2 -10036.024} C_VEL
LIN {X 0,Y 422.022,Z 356.89,A -85,B 0,C 180,E1 -10036.939,E2 -10036.939} C_VEL
LIN {X 0,Y 421.62,Z 368.426,A -85,B 0,C 180,E1 -10037.861,E2 -10037.861} C_VEL
LIN {X 0,Y 421.088,Z 378.634,A -85,B 0,C 180,E1 -10038.874,E2 -10038.874} C_VEL
LIN {X 0,Y 420.428,Z 388.907,A -85,B 0,C 180,E1 -10040.139,E2 -10040.139} C_VEL
LIN {X 0,Y 419.851,Z 397.417,A -85,B 0,C 180,E1 -10041.425,E2 -10041.425} C_VEL
LIN {X 0,Y 419.324,Z 405.26,A -85,B 0,C 180,E1 -10042.888,E2 -10042.888} C_VEL
LIN {X 0,Y 418.967,Z 411.491,A -85,B 0,C 180,E1 -10044.344,E2 -10044.344} C_VEL
LIN {X 0,Y 418.571,Z 416.58,A -85,B 0,C 180,E1 -10045.836,E2 -10045.836} C_VEL
LIN {X 0,Y 418.386,Z 420.823,A -85,B 0,C 180,E1 -10047.484,E2 -10047.484} C_VEL
LIN {X 0,Y 418.215,Z 423.552,A -85,B 0,C 180,E1 -10048.984,E2 -10048.984} C_VEL
LIN {X 0,Y 418.114,Z 425.526,A -85,B 0,C 180,E1 -10050.826,E2 -10050.826} C_VEL
LIN {X 0,Y 418.093,Z 426.017,A -85,B 0,C 180,E1 -10051.922,E2 -10051.922} C_VEL
LIN {X 0,Y 418.122,Z 426.007,A -85,B 0,C 180,E1 -10053.01,E2 -10053.01} C_VEL
LIN {X 0,Y 418.2,Z 425.472,A -85,B 0,C 180,E1 -10054.091,E2 -10054.091} C_VEL
LIN {X 0,Y 418.363,Z 424.476,A -85,B 0,C 180,E1 -10055.167,E2 -10055.167} C_VEL
LIN {X 0,Y 418.525,Z 422.942,A -85,B 0,C 180,E1 -10056.233,E2 -10056.233} C_VEL
LIN {X 0,Y 418.862,Z 419.632,A -85,B 0,C 180,E1 -10057.859,E2 -10057.859} C_VEL
LIN {X 0,Y 419.242,Z 415.327,A -85,B 0,C 180,E1 -10059.388,E2 -10059.388} C_VEL
LIN {X 0,Y 419.749,Z 409.586,A -85,B 0,C 180,E1 -10060.944,E2 -10060.944} C_VEL
LIN {X 0,Y 420.377,Z 402.27,A -85,B 0,C 180,E1 -10062.487,E2 -10062.487} C_VEL
LIN {X 0,Y 420.973,Z 394.783,A -85,B 0,C 180,E1 -10063.762,E2 -10063.762} C_VEL
LIN {X 0,Y 421.624,Z 386.505,A -85,B 0,C 180,E1 -10064.919,E2 -10064.919} C_VEL
LIN {X 0,Y 422.3,Z 376.721,A -85,B 0,C 180,E1 -10066.036,E2 -10066.036} C_VEL
LIN {X 0,Y 422.923,Z 365.843,A -85,B 0,C 180,E1 -10067.036,E2 -10067.036} C_VEL
LIN {X 0,Y 423.25,Z 359.369,A -85,B 0,C 180,E1 -10067.534,E2 -10067.534} C_VEL
LIN {X 0,Y 420.039,Z 348.533,A -85,B 0,C 180,E1 -10068.417,E2 -10068.417} C_VEL
LIN {X 0,Y 418.425,Z 343.963,A -85,B 0,C 180,E1 -10068.802,E2 -10068.802} C_VEL
LIN {X 0,Y 418.323,Z 343.411,A -85,B 0,C 180,E1 -10068.983,E2 -10068.983} C_VEL
LIN {X 0,Y 418.475,Z 343.358,A -85,B 0,C 180,E1 -10072.279,E2 -10072.279} C_VEL
LIN {X 0,Y 418.499,Z 343.355,A -85,B 0,C 180,E1 -10074.217,E2 -10074.217} C_VEL
LIN {X 0,Y 418.531,Z 343.35,A -85,B 0,C 180,E1 -10078.075,E2 -10078.075} C_VEL
LIN {X 0,Y 418.661,Z 343.334,A -85,B 0,C 180,E1 -10080,E2 -10080} C_VEL
LIN {X 0,Y 418.489,Z 343.357,A -85,B 0,C 180,E1 -10082.888,E2 -10082.888} C_VEL
LIN {X 0,Y 418.494,Z 343.355,A -85,B 0,C 180,E1 -10085.783,E2 -10085.783} C_VEL
LIN {X 0,Y 418.368,Z 343.37,A -85,B 0,C 180,E1 -10088.696,E2 -10088.696} C_VEL
LIN {X 0,Y 418.305,Z 343.378,A -85,B 0,C 180,E1 -10091.631,E2 -10091.631} C_VEL
LIN {X 0,Y 418.292,Z 343.38,A -85,B 0,C 180,E1 -10094.597,E2 -10094.597} C_VEL
LIN {X 0,Y 418.27,Z 343.379,A -85,B 0,C 180,E1 -10097.605,E2 -10097.605} C_VEL
LIN {X 0,Y 418.241,Z 343.384,A -85,B 0,C 180,E1 -10100.664,E2 -10100.664} C_VEL
LIN {X 0,Y 418.267,Z 343.38,A -85,B 0,C 180,E1 -10103.783,E2 -10103.783} C_VEL
LIN {X 0,Y 418.303,Z 343.38,A -85,B 0,C 180,E1 -10107.071,E2 -10107.071} C_VEL
LIN {X 0,Y 418.237,Z 343.388,A -85,B 0,C 180,E1 -10110.273,E2 -10110.273} C_VEL
LIN {X 0,Y 418.24,Z 343.386,A -85,B 0,C 180,E1 -10113.678,E2 -10113.678} C_VEL
LIN {X 0,Y 418.232,Z 343.389,A -85,B 0,C 180,E1 -10117.225,E2 -10117.225} C_VEL
LIN {X 0,Y 418.201,Z 343.395,A -85,B 0,C 180,E1 -10120.868,E2 -10120.868} C_VEL
LIN {X 0,Y 418.198,Z 343.393,A -85,B 0,C 180,E1 -10123.729,E2 -10123.729} C_VEL
LIN {X 0,Y 418.197,Z 343.391,A -85,B 0,C 180,E1 -10126.448,E2 -10126.448} C_VEL
LIN {X 0,Y 418.233,Z 343.475,A -85,B 0,C 180,E1 -10127.52,E2 -10127.52} C_VEL
LIN {X 0,Y 419.815,Z 351.292,A -85,B 0,C 180,E1 -10130.496,E2 -10130.496} C_VEL
LIN {X 0,Y 420.87,Z 356.88,A -85,B 0,C 180,E1 -10132.447,E2 -10132.447} C_VEL
LIN {X 0,Y 421.129,Z 360.886,A -85,B 0,C 180,E1 -10133.742,E2 -10133.742} C_VEL
LIN {X 0,Y 419.947,Z 374.024,A -85,B 0,C 180,E1 -10137.621,E2 -10137.621} C_VEL
LIN {X 0,Y 419.153,Z 387.723,A -85,B 0,C 180,E1 -10141.455,E2 -10141.455} C_VEL
LIN {X 0,Y 418.604,Z 399.62,A -85,B 0,C 180,E1 -10144.644,E2 -10144.644} C_VEL
LIN {X 0,Y 418.193,Z 410.836,A -85,B 0,C 180,E1 -10147.565,E2 -10147.565} C_VEL
LIN {X 0,Y 417.88,Z 423.722,A -85,B 0,C 180,E1 -10150.856,E2 -10150.856} C_VEL
LIN {X 0,Y 417.79,Z 430.194,A -85,B 0,C 180,E1 -10152.43,E2 -10152.43} C_VEL
LIN {X 0,Y 418.011,Z 432.65,A -85,B 0,C 180,E1 -10152.551,E2 -10152.551} C_VEL
LIN {X 0,Y 419.653,Z 447.032,A -85,B 0,C 180,E1 -10153.089,E2 -10153.089} C_VEL
LIN {X 0,Y 420.192,Z 460.092,A -85,B 0,C 180,E1 -10153.731,E2 -10153.731} C_VEL
LIN {X 0,Y 420.649,Z 471.963,A -85,B 0,C 180,E1 -10154.496,E2 -10154.496} C_VEL
LIN {X 0,Y 419.764,Z 484.294,A -85,B 0,C 180,E1 -10155.455,E2 -10155.455} C_VEL
LIN {X 0,Y 419.058,Z 495.286,A -85,B 0,C 180,E1 -10156.536,E2 -10156.536} C_VEL
LIN {X 0,Y 418.58,Z 504.487,A -85,B 0,C 180,E1 -10157.639,E2 -10157.639} C_VEL
LIN {X 0,Y 417.989,Z 514.507,A -85,B 0,C 180,E1 -10159.097,E2 -10159.097} C_VEL
LIN {X 0,Y 417.663,Z 522.585,A -85,B 0,C 180,E1 -10160.557,E2 -10160.557} C_VEL
LIN {X 0,Y 417.55,Z 530.095,A -85,B 0,C 180,E1 -10162.262,E2 -10162.262} C_VEL
LIN {X 0,Y 417.528,Z 534.716,A -85,B 0,C 180,E1 -10163.587,E2 -10163.587} C_VEL
LIN {X 0,Y 417.654,Z 539.028,A -85,B 0,C 180,E1 -10165.174,E2 -10165.174} C_VEL
LIN {X 0,Y 417.709,Z 541.04,A -85,B 0,C 180,E1 -10166.141,E2 -10166.141} C_VEL
LIN {X 0,Y 417.679,Z 542.557,A -85,B 0,C 180,E1 -10167.107,E2 -10167.107} C_VEL
LIN {X 0,Y 417.919,Z 544.398,A -85,B 0,C 180,E1 -10169.036,E2 -10169.036} C_VEL
LIN {X 0,Y 417.926,Z 544.648,A -85,B 0,C 180,E1 -10170,E2 -10170} C_VEL
LIN {X 0,Y 417.913,Z 544.465,A -85,B 0,C 180,E1 -10170.964,E2 -10170.964} C_VEL
LIN {X 0,Y 417.654,Z 542.841,A -85,B 0,C 180,E1 -10172.894,E2 -10172.894} C_VEL
LIN {X 0,Y 417.675,Z 541.367,A -85,B 0,C 180,E1 -10173.859,E2 -10173.859} C_VEL
LIN {X 0,Y 417.56,Z 538.304,A -85,B 0,C 180,E1 -10175.311,E2 -10175.311} C_VEL
LIN {X 0,Y 417.522,Z 534.144,A -85,B 0,C 180,E1 -10176.767,E2 -10176.767} C_VEL
LIN {X 0,Y 417.554,Z 527.754,A -85,B 0,C 180,E1 -10178.469,E2 -10178.469} C_VEL
LIN {X 0,Y 417.684,Z 520.778,A -85,B 0,C 180,E1 -10179.931,E2 -10179.931} C_VEL
LIN {X 0,Y 418.158,Z 512.068,A -85,B 0,C 180,E1 -10181.39,E2 -10181.39} C_VEL
LIN {X 0,Y 418.774,Z 503.192,A -85,B 0,C 180,E1 -10182.601,E2 -10182.601} C_VEL
LIN {X 0,Y 419.182,Z 494.614,A -85,B 0,C 180,E1 -10183.575,E2 -10183.575} C_VEL
LIN {X 0,Y 419.766,Z 484.288,A -85,B 0,C 180,E1 -10184.545,E2 -10184.545} C_VEL
LIN {X 0,Y 420.56,Z 473.09,A -85,B 0,C 180,E1 -10185.384,E2 -10185.384} C_VEL
LIN {X 0,Y 420.377,Z 466.07,A -85,B 0,C 180,E1 -10185.826,E2 -10185.826} C_VEL
LIN {X 0,Y 419.586,Z 453.275,A -85,B 0,C 180,E1 -10186.49,E2 -10186.49} C_VEL
LIN {X 0,Y 418.278,Z 439.993,A -85,B 0,C 180,E1 -10186.992,E2 -10186.992} C_VEL
LIN {X 0,Y 417.752,Z 434.766,A -85,B 0,C 180,E1 -10187.175,E2 -10187.175} C_VEL
LIN {X 0,Y 418.063,Z 425.021,A -85,B 0,C 180,E1 -10189.646,E2 -10189.646} C_VEL
LIN {X 0,Y 418.597,Z 411.372,A -85,B 0,C 180,E1 -10193.237,E2 -10193.237} C_VEL
LIN {X 0,Y 419.166,Z 399.618,A -85,B 0,C 180,E1 -10196.379,E2 -10196.379} C_VEL
LIN {X 0,Y 419.841,Z 387.218,A -85,B 0,C 180,E1 -10199.755,E2 -10199.755} C_VEL
LIN {X 0,Y 420.473,Z 377.942,A -85,B 0,C 180,E1 -10202.334,E2 -10202.334} C_VEL
LIN {X 0,Y 421.743,Z 364.097,A -85,B 0,C 180,E1 -10206.268,E2 -10206.268} C_VEL
LIN {X 0,Y 421.539,Z 360.082,A -85,B 0,C 180,E1 -10207.482,E2 -10207.482} C_VEL
LIN {X 0,Y 419.509,Z 349.745,A -85,B 0,C 180,E1 -10210.794,E2 -10210.794} C_VEL
LIN {X 0,Y 418.232,Z 343.451,A -85,B 0,C 180,E1 -10212.982,E2 -10212.982} C_VEL
LIN {X 0,Y 418.199,Z 343.392,A -85,B 0,C 180,E1 -10216.271,E2 -10216.271} C_VEL
LIN {X 0,Y 418.202,Z 343.392,A -85,B 0,C 180,E1 -10219.132,E2 -10219.132} C_VEL
LIN {X 0,Y 418.232,Z 343.386,A -85,B 0,C 180,E1 -10222.775,E2 -10222.775} C_VEL
LIN {X 0,Y 418.24,Z 343.383,A -85,B 0,C 180,E1 -10226.322,E2 -10226.322} C_VEL
LIN {X 0,Y 418.237,Z 343.385,A -85,B 0,C 180,E1 -10229.727,E2 -10229.727} C_VEL
LIN {X 0,Y 418.297,Z 343.381,A -85,B 0,C 180,E1 -10233.022,E2 -10233.022} C_VEL
LIN {X 0,Y 418.265,Z 343.38,A -85,B 0,C 180,E1 -10236.217,E2 -10236.217} C_VEL
LIN {X 0,Y 418.241,Z 343.387,A -85,B 0,C 180,E1 -10239.336,E2 -10239.336} C_VEL
LIN {X 0,Y 418.27,Z 343.38,A -85,B 0,C 180,E1 -10242.395,E2 -10242.395} C_VEL
LIN {X 0,Y 418.292,Z 343.379,A -85,B 0,C 180,E1 -10245.403,E2 -10245.403} C_VEL
LIN {X 0,Y 418.305,Z 343.376,A -85,B 0,C 180,E1 -10248.369,E2 -10248.369} C_VEL
LIN {X 0,Y 418.456,Z 343.357,A -85,B 0,C 180,E1 -10252.278,E2 -10252.278} C_VEL
LIN {X 0,Y 418.494,Z 343.352,A -85,B 0,C 180,E1 -10254.217,E2 -10254.217} C_VEL
LIN {X 0,Y 418.532,Z 343.347,A -85,B 0,C 180,E1 -10258.075,E2 -10258.075} C_VEL
LIN {X 0,Y 418.661,Z 343.331,A -85,B 0,C 180,E1 -10260,E2 -10260} C_VEL
LIN {X 0,Y 418.489,Z 343.358,A -85,B 0,C 180,E1 -10262.888,E2 -10262.888} C_VEL
LIN {X 0,Y 418.481,Z 343.36,A -85,B 0,C 180,E1 -10266.751,E2 -10266.751} C_VEL
LIN {X 0,Y 418.332,Z 343.372,A -85,B 0,C 180,E1 -10269.672,E2 -10269.672} C_VEL
LIN {X 0,Y 418.337,Z 343.374,A -85,B 0,C 180,E1 -10273.001,E2 -10273.001} C_VEL
LIN {X 0,Y 418.304,Z 343.38,A -85,B 0,C 180,E1 -10276.736,E2 -10276.736} C_VEL
LIN {X 0,Y 418.263,Z 343.381,A -85,B 0,C 180,E1 -10279.791,E2 -10279.791} C_VEL
LIN {X 0,Y 418.231,Z 343.389,A -85,B 0,C 180,E1 -10282.737,E2 -10282.737} C_VEL
LIN {X 0,Y 418.263,Z 343.382,A -85,B 0,C 180,E1 -10285.905,E2 -10285.905} C_VEL
LIN {X 0,Y 418.267,Z 343.38,A -85,B 0,C 180,E1 -10289.162,E2 -10289.162} C_VEL
LIN {X 0,Y 418.251,Z 343.384,A -85,B 0,C 180,E1 -10292.845,E2 -10292.845} C_VEL
LIN {X 0,Y 418.242,Z 343.39,A -85,B 0,C 180,E1 -10296.239,E2 -10296.239} C_VEL
LIN {X 0,Y 418.258,Z 343.382,A -85,B 0,C 180,E1 -10299.681,E2 -10299.681} C_VEL
LIN {X 0,Y 418.24,Z 343.389,A -85,B 0,C 180,E1 -10302.324,E2 -10302.324} C_VEL
LIN {X 0,Y 418.235,Z 343.384,A -85,B 0,C 180,E1 -10305.11,E2 -10305.11} C_VEL
LIN {X 0,Y 418.253,Z 343.385,A -85,B 0,C 180,E1 -10307.77,E2 -10307.77} C_VEL
LIN {X 0,Y 418.258,Z 343.383,A -85,B 0,C 180,E1 -10311.56,E2 -10311.56} C_VEL
LIN {X 0,Y 418.258,Z 343.381,A -85,B 0,C 180,E1 -10315.16,E2 -10315.16} C_VEL
LIN {X 0,Y 418.247,Z 343.384,A -85,B 0,C 180,E1 -10317.473,E2 -10317.473} C_VEL
LIN {X 0,Y 418.276,Z 343.379,A -85,B 0,C 180,E1 -10320.894,E2 -10320.894} C_VEL
LIN {X 0,Y 418.271,Z 343.384,A -85,B 0,C 180,E1 -10324.097,E2 -10324.097} C_VEL
LIN {X 0,Y 418.239,Z 343.384,A -85,B 0,C 180,E1 -10327.265,E2 -10327.265} C_VEL
LIN {X 0,Y 418.284,Z 343.379,A -85,B 0,C 180,E1 -10330.365,E2 -10330.365} C_VEL
LIN {X 0,Y 418.328,Z 343.375,A -85,B 0,C 180,E1 -10333.405,E2 -10333.405} C_VEL
LIN {X 0,Y 418.348,Z 343.37,A -85,B 0,C 180,E1 -10336.999,E2 -10336.999} C_VEL
LIN {X 0,Y 418.344,Z 343.371,A -85,B 0,C 180,E1 -10340.329,E2 -10340.329} C_VEL
LIN {X 0,Y 418.497,Z 343.354,A -85,B 0,C 180,E1 -10343.249,E2 -10343.249} C_VEL
LIN {X 0,Y 418.344,Z 343.373,A -85,B 0,C 180,E1 -10345.182,E2 -10345.182} C_VEL
LIN {X 0,Y 418.547,Z 343.347,A -85,B 0,C 180,E1 -10348.076,E2 -10348.076} C_VEL
LIN {X 0,Y 418.676,Z 343.331,A -85,B 0,C 180,E1 -10350,E2 -10350} C_VEL
LIN {X 0,Y 418.514,Z 343.35,A -85,B 0,C 180,E1 -10352.888,E2 -10352.888} C_VEL
LIN {X 0,Y 418.49,Z 343.353,A -85,B 0,C 180,E1 -10356.751,E2 -10356.751} C_VEL
LIN {X 0,Y 418.343,Z 343.374,A -85,B 0,C 180,E1 -10359.671,E2 -10359.671} C_VEL
LIN {X 0,Y 418.348,Z 343.373,A -85,B 0,C 180,E1 -10363.001,E2 -10363.001} C_VEL
LIN {X 0,Y 418.324,Z 343.376,A -85,B 0,C 180,E1 -10363.349,E2 -10363.349} C_VEL
LIN {X 0,Y 417.632,Z 343.464,A -85,B 0,C 180,E1 -10364.153,E2 -10364.153} C_VEL
LIN {X 0,Y 414.753,Z 343.823,A -85,B 0,C 180,E1 -10365.458,E2 -10365.458} C_VEL
LIN {X 0,Y 412.339,Z 344.12,A -85,B 0,C 180,E1 -10366.512,E2 -10366.512} C_VEL
LIN {X 0,Y 411.317,Z 344.253,A -85,B 0,C 180,E1 -10367.327,E2 -10367.327} C_VEL
LIN {X 0,Y 411.241,Z 344.255,A -85,B 0,C 180,E1 -10367.603,E2 -10367.603} C_VEL
LIN {X 0,Y 411.198,Z 344.265,A -85,B 0,C 180,E1 -10371.033,E2 -10371.033} C_VEL
LIN {X 0,Y 411.227,Z 344.257,A -85,B 0,C 180,E1 -10374.215,E2 -10374.215} C_VEL
LIN {X 0,Y 411.258,Z 344.256,A -85,B 0,C 180,E1 -10377.477,E2 -10377.477} C_VEL
LIN {X 0,Y 411.188,Z 344.266,A -85,B 0,C 180,E1 -10380.847,E2 -10380.847} C_VEL
LIN {X 0,Y 411.204,Z 344.26,A -85,B 0,C 180,E1 -10384.333,E2 -10384.333} C_VEL
LIN {X 0,Y 411.203,Z 344.26,A -85,B 0,C 180,E1 -10387.972,E2 -10387.972} C_VEL
LIN {X 0,Y 411.207,Z 344.266,A -85,B 0,C 180,E1 -10391.235,E2 -10391.235} C_VEL
LIN {X 0,Y 411.229,Z 344.263,A -85,B 0,C 180,E1 -10394.482,E2 -10394.482} C_VEL
LIN {X 0,Y 411.288,Z 344.501,A -85,B 0,C 180,E1 -10395.625,E2 -10395.625} C_VEL
LIN {X 0,Y 411.662,Z 345.955,A -85,B 0,C 180,E1 -10395.809,E2 -10395.809} C_VEL
LIN {X 0,Y 415.232,Z 358.902,A -85,B 0,C 180,E1 -10396.809,E2 -10396.809} C_VEL
LIN {X 0,Y 414.685,Z 370.149,A -85,B 0,C 180,E1 -10397.733,E2 -10397.733} C_VEL
LIN {X 0,Y 414.083,Z 381.155,A -85,B 0,C 180,E1 -10398.877,E2 -10398.877} C_VEL
LIN {X 0,Y 413.429,Z 390.973,A -85,B 0,C 180,E1 -10400.134,E2 -10400.134} C_VEL
LIN {X 0,Y 412.836,Z 399.844,A -85,B 0,C 180,E1 -10401.542,E2 -10401.542} C_VEL
LIN {X 0,Y 412.303,Z 407.487,A -85,B 0,C 180,E1 -10403.051,E2 -10403.051} C_VEL
LIN {X 0,Y 411.87,Z 413.534,A -85,B 0,C 180,E1 -10404.538,E2 -10404.538} C_VEL
LIN {X 0,Y 411.598,Z 417.364,A -85,B 0,C 180,E1 -10405.704,E2 -10405.704} C_VEL
LIN {X 0,Y 411.361,Z 421.808,A -85,B 0,C 180,E1 -10407.441,E2 -10407.441} C_VEL
LIN {X 0,Y 411.173,Z 424.823,A -85,B 0,C 180,E1 -10409.151,E2 -10409.151} C_VEL
LIN {X 0,Y 411.101,Z 426.439,A -85,B 0,C 180,E1 -10410.675,E2 -10410.675} C_VEL
LIN {X 0,Y 411.075,Z 427.089,A -85,B 0,C 180,E1 -10412.509,E2 -10412.509} C_VEL
LIN {X 0,Y 411.149,Z 426.841,A -85,B 0,C 180,E1 -10413.613,E2 -10413.613} C_VEL
LIN {X 0,Y 411.321,Z 425.871,A -85,B 0,C 180,E1 -10414.898,E2 -10414.898} C_VEL
LIN {X 0,Y 411.45,Z 424.803,A -85,B 0,C 180,E1 -10415.799,E2 -10415.799} C_VEL
LIN {X 0,Y 411.733,Z 422.457,A -85,B 0,C 180,E1 -10417.179,E2 -10417.179} C_VEL
LIN {X 0,Y 412.144,Z 418.001,A -85,B 0,C 180,E1 -10419.017,E2 -10419.017} C_VEL
LIN {X 0,Y 412.676,Z 412.678,A -85,B 0,C 180,E1 -10420.604,E2 -10420.604} C_VEL
LIN {X 0,Y 413.344,Z 405.811,A -85,B 0,C 180,E1 -10422.2,E2 -10422.2} C_VEL
LIN {X 0,Y 413.923,Z 399.009,A -85,B 0,C 180,E1 -10423.477,E2 -10423.477} C_VEL
LIN {X 0,Y 414.595,Z 391.015,A -85,B 0,C 180,E1 -10424.711,E2 -10424.711} C_VEL
LIN {X 0,Y 415.353,Z 381.324,A -85,B 0,C 180,E1 -10425.923,E2 -10425.923} C_VEL
LIN {X 0,Y 416.07,Z 369.958,A -85,B 0,C 180,E1 -10427.067,E2 -10427.067} C_VEL
LIN {X 0,Y 416.484,Z 360.618,A -85,B 0,C 180,E1 -10427.823,E2 -10427.823} C_VEL
LIN {X 0,Y 413.205,Z 350.004,A -85,B 0,C 180,E1 -10428.72,E2 -10428.72} C_VEL
LIN {X 0,Y 411.423,Z 344.982,A -85,B 0,C 180,E1 -10429.138,E2 -10429.138} C_VEL
LIN {X 0,Y 411.31,Z 344.283,A -85,B 0,C 180,E1 -10429.353,E2 -10429.353} C_VEL
LIN {X 0,Y 411.444,Z 344.235,A -85,B 0,C 180,E1 -10433.133,E2 -10433.133} C_VEL
LIN {X 0,Y 411.297,Z 344.252,A -85,B 0,C 180,E1 -10435.099,E2 -10435.099} C_VEL
LIN {X 0,Y 411.5,Z 344.227,A -85,B 0,C 180,E1 -10438.043,E2 -10438.043} C_VEL
LIN {X 0,Y 411.631,Z 344.21,A -85,B 0,C 180,E1 -10440,E2 -10440} C_VEL
LIN {X 0,Y 411.446,Z 344.235,A -85,B 0,C 180,E1 -10442.937,E2 -10442.937} C_VEL
LIN {X 0,Y 411.455,Z 344.231,A -85,B 0,C 180,E1 -10445.882,E2 -10445.882} C_VEL
LIN {X 0,Y 411.309,Z 344.25,A -85,B 0,C 180,E1 -10448.846,E2 -10448.846} C_VEL
LIN {X 0,Y 411.274,Z 344.252,A -85,B 0,C 180,E1 -10451.833,E2 -10451.833} C_VEL
LIN {X 0,Y 411.25,Z 344.26,A -85,B 0,C 180,E1 -10454.853,E2 -10454.853} C_VEL
LIN {X 0,Y 411.236,Z 344.254,A -85,B 0,C 180,E1 -10457.916,E2 -10457.916} C_VEL
LIN {X 0,Y 411.187,Z 344.263,A -85,B 0,C 180,E1 -10461.035,E2 -10461.035} C_VEL
LIN {X 0,Y 411.211,Z 344.259,A -85,B 0,C 180,E1 -10464.216,E2 -10464.216} C_VEL
LIN {X 0,Y 411.251,Z 344.258,A -85,B 0,C 180,E1 -10467.478,E2 -10467.478} C_VEL
